LIN {X 0,Y 411.168,Z 328.267,A -85,B 0,C 180,E1 -10479.721,E2 -10479.721} C_VEL
LIN {X 0,Y 411.16,Z 328.272,A -85,B 0,C 180,E1 -10483.136,E2 -10483.136} C_VEL
LIN {X 0,Y 411.167,Z 328.27,A -85,B 0,C 180,E1 -10485.881,E2 -10485.881} C_VEL
LIN {X 0,Y 411.213,Z 328.29,A -85,B 0,C 180,E1 -10488.764,E2 -10488.764} C_VEL
LIN {X 0,Y 412.183,Z 333.965,A -85,B 0,C 180,E1 -10492.134,E2 -10492.134} C_VEL
LIN {X 0,Y 412.545,Z 338.866,A -85,B 0,C 180,E1 -10494.857,E2 -10494.857} C_VEL
LIN {X 0,Y 412.139,Z 345.061,A -85,B 0,C 180,E1 -10498.087,E2 -10498.087} C_VEL
LIN {X 0,Y 411.71,Z 351.771,A -85,B 0,C 180,E1 -10501.447,E2 -10501.447} C_VEL
LIN {X 0,Y 411.267,Z 358.916,A -85,B 0,C 180,E1 -10504.918,E2 -10504.918} C_VEL
LIN {X 0,Y 410.904,Z 366.234,A -85,B 0,C 180,E1 -10508.424,E2 -10508.424} C_VEL
LIN {X 0,Y 410.611,Z 372.815,A -85,B 0,C 180,E1 -10511.54,E2 -10511.54} C_VEL
LIN {X 0,Y 410.564,Z 374.685,A -85,B 0,C 180,E1 -10512.421,E2 -10512.421} C_VEL
LIN {X 0,Y 412.967,Z 388.008,A -85,B 0,C 180,E1 -10512.93,E2 -10512.93} C_VEL
LIN {X 0,Y 414.869,Z 400.705,A -85,B 0,C 180,E1 -10513.605,E2 -10513.605} C_VEL
LIN {X 0,Y 414.575,Z 409.621,A -85,B 0,C 180,E1 -10514.141,E2 -10514.141} C_VEL
LIN {X 0,Y 413.832,Z 420.921,A -85,B 0,C 180,E1 -10514.99,E2 -10514.99} C_VEL
LIN {X 0,Y 413.057,Z 432.111,A -85,B 0,C 180,E1 -10516.055,E2 -10516.055} C_VEL
LIN {X 0,Y 412.36,Z 441.79,A -85,B 0,C 180,E1 -10517.199,E2 -10517.199} C_VEL
LIN {X 0,Y 411.629,Z 450.278,A -85,B 0,C 180,E1 -10518.427,E2 -10518.427} C_VEL
LIN {X 0,Y 411.026,Z 458.564,A -85,B 0,C 180,E1 -10519.906,E2 -10519.906} C_VEL
LIN {X 0,Y 410.576,Z 465.244,A -85,B 0,C 180,E1 -10521.386,E2 -10521.386} C_VEL
LIN {X 0,Y 410.253,Z 471.36,A -85,B 0,C 180,E1 -10523.112,E2 -10523.112} C_VEL
LIN {X 0,Y 410.065,Z 475.333,A -85,B 0,C 180,E1 -10524.591,E2 -10524.591} C_VEL
LIN {X 0,Y 409.943,Z 478.268,A -85,B 0,C 180,E1 -10526.067,E2 -10526.067} C_VEL
LIN {X 0,Y 409.963,Z 480.666,A -85,B 0,C 180,E1 -10528.035,E2 -10528.035} C_VEL
LIN {X 0,Y 409.919,Z 481.275,A -85,B 0,C 180,E1 -10529.017,E2 -10529.017} C_VEL
LIN {X 0,Y 409.888,Z 481.491,A -85,B 0,C 180,E1 -10530,E2 -10530} C_VEL
LIN {X 0,Y 409.918,Z 481.275,A -85,B 0,C 180,E1 -10530.982,E2 -10530.982} C_VEL
LIN {X 0,Y 409.963,Z 480.669,A -85,B 0,C 180,E1 -10531.964,E2 -10531.964} C_VEL
LIN {X 0,Y 409.943,Z 478.274,A -85,B 0,C 180,E1 -10533.932,E2 -10533.932} C_VEL
LIN {X 0,Y 410.063,Z 475.336,A -85,B 0,C 180,E1 -10535.408,E2 -10535.408} C_VEL
LIN {X 0,Y 410.198,Z 471.359,A -85,B 0,C 180,E1 -10536.888,E2 -10536.888} C_VEL
LIN {X 0,Y 410.575,Z 465.247,A -85,B 0,C 180,E1 -10538.613,E2 -10538.613} C_VEL
LIN {X 0,Y 411.025,Z 458.568,A -85,B 0,C 180,E1 -10540.093,E2 -10540.093} C_VEL
LIN {X 0,Y 411.633,Z 450.282,A -85,B 0,C 180,E1 -10541.572,E2 -10541.572} C_VEL
LIN {X 0,Y 412.375,Z 441.796,A -85,B 0,C 180,E1 -10542.8,E2 -10542.8} C_VEL
LIN {X 0,Y 413.08,Z 431.211,A -85,B 0,C 180,E1 -10544.04,E2 -10544.04} C_VEL
LIN {X 0,Y 413.891,Z 419.499,A -85,B 0,C 180,E1 -10545.133,E2 -10545.133} C_VEL
LIN {X 0,Y 414.716,Z 407.771,A -85,B 0,C 180,E1 -10545.975,E2 -10545.975} C_VEL
LIN {X 0,Y 414.824,Z 400.648,A -85,B 0,C 180,E1 -10546.399,E2 -10546.399} C_VEL
LIN {X 0,Y 412.854,Z 387.284,A -85,B 0,C 180,E1 -10547.101,E2 -10547.101} C_VEL
LIN {X 0,Y 410.564,Z 374.685,A -85,B 0,C 180,E1 -10547.578,E2 -10547.578} C_VEL
LIN {X 0,Y 410.855,Z 367.344,A -85,B 0,C 180,E1 -10551.051,E2 -10551.051} C_VEL
LIN {X 0,Y 411.168,Z 360.704,A -85,B 0,C 180,E1 -10554.218,E2 -10554.218} C_VEL
LIN {X 0,Y 411.55,Z 353.989,A -85,B 0,C 180,E1 -10557.455,E2 -10557.455} C_VEL
LIN {X 0,Y 411.993,Z 347.272,A -85,B 0,C 180,E1 -10560.78,E2 -10560.78} C_VEL
LIN {X 0,Y 412.444,Z 340.595,A -85,B 0,C 180,E1 -10564.215,E2 -10564.215} C_VEL
LIN {X 0,Y 412.503,Z 337.275,A -85,B 0,C 180,E1 -10565.999,E2 -10565.999} C_VEL
LIN {X 0,Y 412.086,Z 333.137,A -85,B 0,C 180,E1 -10568.324,E2 -10568.324} C_VEL
LIN {X 0,Y 411.243,Z 328.265,A -85,B 0,C 180,E1 -10571.241,E2 -10571.241} C_VEL
LIN {X 0,Y 411.223,Z 328.263,A -85,B 0,C 180,E1 -10574.482,E2 -10574.482} C_VEL
LIN {X 0,Y 411.157,Z 328.268,A -85,B 0,C 180,E1 -10578.192,E2 -10578.192} C_VEL
LIN {X 0,Y 411.193,Z 328.263,A -85,B 0,C 180,E1 -10581.832,E2 -10581.832} C_VEL
LIN {X 0,Y 411.204,Z 328.264,A -85,B 0,C 180,E1 -10585.121,E2 -10585.121} C_VEL
LIN {X 0,Y 411.158,Z 328.269,A -85,B 0,C 180,E1 -10588.002,E2 -10588.002} C_VEL
LIN {X 0,Y 411.171,Z 328.265,A -85,B 0,C 180,E1 -10591.406,E2 -10591.406} C_VEL
LIN {X 0,Y 411.218,Z 328.261,A -85,B 0,C 180,E1 -10594.929,E2 -10594.929} C_VEL
LIN {X 0,Y 411.196,Z 328.265,A -85,B 0,C 180,E1 -10597.913,E2 -10597.913} C_VEL
LIN {X 0,Y 411.215,Z 328.261,A -85,B 0,C 180,E1 -10601.051,E2 -10601.051} C_VEL
LIN {X 0,Y 411.244,Z 328.261,A -85,B 0,C 180,E1 -10604.131,E2 -10604.131} C_VEL
LIN {X 0,Y 411.293,Z 328.25,A -85,B 0,C 180,E1 -10607.165,E2 -10607.165} C_VEL
LIN {X 0,Y 411.283,Z 328.255,A -85,B 0,C 180,E1 -10610.161,E2 -10610.161} C_VEL
LIN {X 0,Y 411.453,Z 328.231,A -85,B 0,C 180,E1 -10613.133,E2 -10613.133} C_VEL
LIN {X 0,Y 411.309,Z 328.249,A -85,B 0,C 180,E1 -10615.099,E2 -10615.099} C_VEL
LIN {X 0,Y 411.502,Z 328.228,A -85,B 0,C 180,E1 -10618.043,E2 -10618.043} C_VEL
LIN {X 0,Y 411.622,Z 328.212,A -85,B 0,C 180,E1 -10620,E2 -10620} C_VEL
LIN {X 0,Y 411.449,Z 328.231,A -85,B 0,C 180,E1 -10622.937,E2 -10622.937} C_VEL
LIN {X 0,Y 411.452,Z 328.232,A -85,B 0,C 180,E1 -10626.867,E2 -10626.867} C_VEL
LIN {X 0,Y 411.283,Z 328.254,A -85,B 0,C 180,E1 -10629.839,E2 -10629.839} C_VEL
LIN {X 0,Y 411.295,Z 328.253,A -85,B 0,C 180,E1 -10633.104,E2 -10633.104} C_VEL
LIN {X 0,Y 411.248,Z 328.258,A -85,B 0,C 180,E1 -10636.889,E2 -10636.889} C_VEL
LIN {X 0,Y 411.222,Z 328.259,A -85,B 0,C 180,E1 -10639.987,E2 -10639.987} C_VEL
LIN {X 0,Y 411.193,Z 328.267,A -85,B 0,C 180,E1 -10643.148,E2 -10643.148} C_VEL
LIN {X 0,Y 411.177,Z 328.266,A -85,B 0,C 180,E1 -10646.385,E2 -10646.385} C_VEL
LIN {X 0,Y 411.189,Z 328.263,A -85,B 0,C 180,E1 -10649.714,E2 -10649.714} C_VEL
LIN {X 0,Y 411.199,Z 328.265,A -85,B 0,C 180,E1 -10653.157,E2 -10653.157} C_VEL
LIN {X 0,Y 411.186,Z 328.268,A -85,B 0,C 180,E1 -10656.553,E2 -10656.553} C_VEL
LIN {X 0,Y 411.163,Z 328.267,A -85,B 0,C 180,E1 -10659.721,E2 -10659.721} C_VEL
LIN {X 0,Y 411.158,Z 328.268,A -85,B 0,C 180,E1 -10663.136,E2 -10663.136} C_VEL
LIN {X 0,Y 411.163,Z 328.267,A -85,B 0,C 180,E1 -10665.882,E2 -10665.882} C_VEL
LIN {X 0,Y 411.197,Z 328.265,A -85,B 0,C 180,E1 -10668.767,E2 -10668.767} C_VEL
LIN {X 0,Y 411.193,Z 328.267,A -85,B 0,C 180,E1 -10672.028,E2 -10672.028} C_VEL
LIN {X 0,Y 411.147,Z 328.274,A -85,B 0,C 180,E1 -10673.457,E2 -10673.457} C_VEL
LIN {X 0,Y 411.083,Z 328.68,A -85,B 0,C 180,E1 -10674.461,E2 -10674.461} C_VEL
LIN {X 0,Y 411.069,Z 331.626,A -85,B 0,C 180,E1 -10676.903,E2 -10676.903} C_VEL
LIN {X 0,Y 410.849,Z 335.82,A -85,B 0,C 180,E1 -10680.26,E2 -10680.26} C_VEL
LIN {X 0,Y 410.661,Z 340.084,A -85,B 0,C 180,E1 -10683.58,E2 -10683.58} C_VEL
LIN {X 0,Y 410.515,Z 344.369,A -85,B 0,C 180,E1 -10686.812,E2 -10686.812} C_VEL
LIN {X 0,Y 410.383,Z 349.289,A -85,B 0,C 180,E1 -10690.374,E2 -10690.374} C_VEL
LIN {X 0,Y 410.314,Z 352.471,A -85,B 0,C 180,E1 -10692.493,E2 -10692.493} C_VEL
LIN {X 0,Y 413.528,Z 365.928,A -85,B 0,C 180,E1 -10693.083,E2 -10693.083} C_VEL
LIN {X 0,Y 415.374,Z 375.743,A -85,B 0,C 180,E1 -10693.63,E2 -10693.63} C_VEL
LIN {X 0,Y 414.752,Z 388.201,A -85,B 0,C 180,E1 -10694.396,E2 -10694.396} C_VEL
LIN {X 0,Y 414.048,Z 398.961,A -85,B 0,C 180,E1 -10695.25,E2 -10695.25} C_VEL
LIN {X 0,Y 413.36,Z 409.923,A -85,B 0,C 180,E1 -10696.356,E2 -10696.356} C_VEL
LIN {X 0,Y 412.474,Z 420.598,A -85,B 0,C 180,E1 -10697.703,E2 -10697.703} C_VEL
LIN {X 0,Y 411.863,Z 428.466,A -85,B 0,C 180,E1 -10698.933,E2 -10698.933} C_VEL
LIN {X 0,Y 411.231,Z 436.156,A -85,B 0,C 180,E1 -10700.409,E2 -10700.409} C_VEL
LIN {X 0,Y 410.669,Z 443.213,A -85,B 0,C 180,E1 -10702.132,E2 -10702.132} C_VEL
LIN {X 0,Y 410.4,Z 447.969,A -85,B 0,C 180,E1 -10703.63,E2 -10703.63} C_VEL
LIN {X 0,Y 410.172,Z 451.508,A -85,B 0,C 180,E1 -10705.086,E2 -10705.086} C_VEL
LIN {X 0,Y 410.063,Z 453.368,A -85,B 0,C 180,E1 -10706.069,E2 -10706.069} C_VEL
LIN {X 0,Y 410.062,Z 454.765,A -85,B 0,C 180,E1 -10707.053,E2 -10707.053} C_VEL
LIN {X 0,Y 410.013,Z 455.761,A -85,B 0,C 180,E1 -10708.036,E2 -10708.036} C_VEL
LIN {X 0,Y 409.927,Z 456.609,A -85,B 0,C 180,E1 -10710,E2 -10710} C_VEL
LIN {X 0,Y 409.939,Z 456.42,A -85,B 0,C 180,E1 -10710.983,E2 -10710.983} C_VEL
LIN {X 0,Y 410.013,Z 455.835,A -85,B 0,C 180,E1 -10711.965,E2 -10711.965} C_VEL
LIN {X 0,Y 410.061,Z 454.869,A -85,B 0,C 180,E1 -10712.948,E2 -10712.948} C_VEL
LIN {X 0,Y 410.06,Z 453.516,A -85,B 0,C 180,E1 -10713.931,E2 -10713.931} C_VEL
LIN {X 0,Y 410.277,Z 450.65,A -85,B 0,C 180,E1 -10715.406,E2 -10715.406} C_VEL
LIN {X 0,Y 410.463,Z 446.768,A -85,B 0,C 180,E1 -10716.884,E2 -10716.884} C_VEL
LIN {X 0,Y 410.801,Z 441.757,A -85,B 0,C 180,E1 -10718.362,E2 -10718.362} C_VEL
LIN {X 0,Y 410.999,Z 439.011,A -85,B 0,C 180,E1 -10719.045,E2 -10719.045} C_VEL
LIN {X 0,Y 410.59,Z 436.033,A -85,B 0,C 180,E1 -10719.756,E2 -10719.756} C_VEL
LIN {X 0,Y 408.194,Z 430.826,A -85,B 0,C 180,E1 -10720.891,E2 -10720.891} C_VEL
LIN {X 0,Y 405.855,Z 424.967,A -85,B 0,C 180,E1 -10721.971,E2 -10721.971} C_VEL
LIN {X 0,Y 405.532,Z 420.966,A -85,B 0,C 180,E1 -10722.585,E2 -10722.585} C_VEL
LIN {X 0,Y 406.417,Z 410.939,A -85,B 0,C 180,E1 -10723.883,E2 -10723.883} C_VEL
LIN {X 0,Y 407.113,Z 400.203,A -85,B 0,C 180,E1 -10725.008,E2 -10725.008} C_VEL
LIN {X 0,Y 407.831,Z 389.733,A -85,B 0,C 180,E1 -10725.877,E2 -10725.877} C_VEL
LIN {X 0,Y 408.532,Z 377.621,A -85,B 0,C 180,E1 -10726.654,E2 -10726.654} C_VEL
LIN {X 0,Y 406.637,Z 367.045,A -85,B 0,C 180,E1 -10727.273,E2 -10727.273} C_VEL
LIN {X 0,Y 403.47,Z 354.02,A -85,B 0,C 180,E1 -10727.875,E2 -10727.875} C_VEL
LIN {X 0,Y 403.203,Z 352.513,A -85,B 0,C 180,E1 -10727.947,E2 -10727.947} C_VEL
LIN {X 0,Y 403.313,Z 349.051,A -85,B 0,C 180,E1 -10730.396,E2 -10730.396} C_VEL
LIN {X 0,Y 403.454,Z 344.71,A -85,B 0,C 180,E1 -10733.619,E2 -10733.619} C_VEL
LIN {X 0,Y 403.666,Z 340.39,A -85,B 0,C 180,E1 -10736.915,E2 -10736.915} C_VEL
LIN {X 0,Y 403.846,Z 336.129,A -85,B 0,C 180,E1 -10740.31,E2 -10740.31} C_VEL
LIN {X 0,Y 404.05,Z 332.333,A -85,B 0,C 180,E1 -10743.394,E2 -10743.394} C_VEL
LIN {X 0,Y 404.099,Z 330.186,A -85,B 0,C 180,E1 -10745.173,E2 -10745.173} C_VEL
LIN {X 0,Y 404.063,Z 329.158,A -85,B 0,C 180,E1 -10746.254,E2 -10746.254} C_VEL
LIN {X 0,Y 404.149,Z 329.146,A -85,B 0,C 180,E1 -10748.757,E2 -10748.757} C_VEL
LIN {X 0,Y 404.123,Z 329.148,A -85,B 0,C 180,E1 -10751.599,E2 -10751.599} C_VEL
LIN {X 0,Y 404.145,Z 329.14,A -85,B 0,C 180,E1 -10754.522,E2 -10754.522} C_VEL
LIN {X 0,Y 404.119,Z 329.147,A -85,B 0,C 180,E1 -10757.293,E2 -10757.293} C_VEL
LIN {X 0,Y 404.131,Z 329.144,A -85,B 0,C 180,E1 -10759.951,E2 -10759.951} C_VEL
LIN {X 0,Y 404.134,Z 329.146,A -85,B 0,C 180,E1 -10763.125,E2 -10763.125} C_VEL
LIN {X 0,Y 404.143,Z 329.141,A -85,B 0,C 180,E1 -10766.187,E2 -10766.187} C_VEL
LIN {X 0,Y 404.141,Z 329.142,A -85,B 0,C 180,E1 -10769.714,E2 -10769.714} C_VEL
LIN {X 0,Y 404.122,Z 329.148,A -85,B 0,C 180,E1 -10773.117,E2 -10773.117} C_VEL
LIN {X 0,Y 404.158,Z 329.14,A -85,B 0,C 180,E1 -10776.425,E2 -10776.425} C_VEL
LIN {X 0,Y 404.188,Z 329.135,A -85,B 0,C 180,E1 -10779.874,E2 -10779.874} C_VEL
LIN {X 0,Y 404.213,Z 329.136,A -85,B 0,C 180,E1 -10782.993,E2 -10782.993} C_VEL
LIN {X 0,Y 404.279,Z 329.127,A -85,B 0,C 180,E1 -10786.939,E2 -10786.939} C_VEL
LIN {X 0,Y 404.254,Z 329.128,A -85,B 0,C 180,E1 -10789.988,E2 -10789.988} C_VEL
LIN {X 0,Y 404.408,Z 329.11,A -85,B 0,C 180,E1 -10793.013,E2 -10793.013} C_VEL
LIN {X 0,Y 404.28,Z 329.125,A -85,B 0,C 180,E1 -10795.013,E2 -10795.013} C_VEL
LIN {X 0,Y 404.475,Z 329.101,A -85,B 0,C 180,E1 -10798.008,E2 -10798.008} C_VEL
LIN {X 0,Y 404.595,Z 329.087,A -85,B 0,C 180,E1 -10800,E2 -10800} C_VEL
LIN {X 0,Y 404.411,Z 329.108,A -85,B 0,C 180,E1 -10802.988,E2 -10802.988} C_VEL
LIN {X 0,Y 404.42,Z 329.111,A -85,B 0,C 180,E1 -10805.985,E2 -10805.985} C_VEL
LIN {X 0,Y 404.287,Z 329.123,A -85,B 0,C 180,E1 -10809.001,E2 -10809.001} C_VEL
LIN {X 0,Y 404.252,Z 329.133,A -85,B 0,C 180,E1 -10812.042,E2 -10812.042} C_VEL
LIN {X 0,Y 404.199,Z 329.134,A -85,B 0,C 180,E1 -10815.118,E2 -10815.118} C_VEL
LIN {X 0,Y 404.206,Z 329.136,A -85,B 0,C 180,E1 -10818.238,E2 -10818.238} C_VEL
LIN {X 0,Y 404.135,Z 329.145,A -85,B 0,C 180,E1 -10821.42,E2 -10821.42} C_VEL
LIN {X 0,Y 404.163,Z 329.138,A -85,B 0,C 180,E1 -10824.667,E2 -10824.667} C_VEL
LIN {X 0,Y 404.116,Z 329.146,A -85,B 0,C 180,E1 -10828.006,E2 -10828.006} C_VEL
LIN {X 0,Y 404.14,Z 329.142,A -85,B 0,C 180,E1 -10830.286,E2 -10830.286} C_VEL
LIN {X 0,Y 404.143,Z 329.144,A -85,B 0,C 180,E1 -10833.813,E2 -10833.813} C_VEL
LIN {X 0,Y 404.136,Z 329.144,A -85,B 0,C 180,E1 -10836.876,E2 -10836.876} C_VEL
LIN {X 0,Y 404.115,Z 329.144,A -85,B 0,C 180,E1 -10840.075,E2 -10840.075} C_VEL
LIN {X 0,Y 404.14,Z 329.147,A -85,B 0,C 180,E1 -10843.082,E2 -10843.082} C_VEL
LIN {X 0,Y 404.147,Z 329.145,A -85,B 0,C 180,E1 -10845.926,E2 -10845.926} C_VEL
LIN {X 0,Y 404.169,Z 329.157,A -85,B 0,C 180,E1 -10848.476,E2 -10848.476} C_VEL
LIN {X 0,Y 404.99,Z 333.851,A -85,B 0,C 180,E1 -10851.344,E2 -10851.344} C_VEL
LIN {X 0,Y 405.502,Z 338.276,A -85,B 0,C 180,E1 -10853.895,E2 -10853.895} C_VEL
LIN {X 0,Y 405.331,Z 342.775,A -85,B 0,C 180,E1 -10856.333,E2 -10856.333} C_VEL
LIN {X 0,Y 404.905,Z 349.379,A -85,B 0,C 180,E1 -10859.778,E2 -10859.778} C_VEL
LIN {X 0,Y 404.427,Z 356.085,A -85,B 0,C 180,E1 -10863.14,E2 -10863.14} C_VEL
LIN {X 0,Y 404.036,Z 362.738,A -85,B 0,C 180,E1 -10866.417,E2 -10866.417} C_VEL
LIN {X 0,Y 403.676,Z 370.283,A -85,B 0,C 180,E1 -10870.076,E2 -10870.076} C_VEL
LIN {X 0,Y 403.508,Z 374.603,A -85,B 0,C 180,E1 -10872.107,E2 -10872.107} C_VEL
LIN {X 0,Y 405.943,Z 387.743,A -85,B 0,C 180,E1 -10872.624,E2 -10872.624} C_VEL
LIN {X 0,Y 407.939,Z 401.142,A -85,B 0,C 180,E1 -10873.356,E2 -10873.356} C_VEL
LIN {X 0,Y 407.839,Z 407.78,A -85,B 0,C 180,E1 -10873.761,E2 -10873.761} C_VEL
LIN {X 0,Y 407.063,Z 419.278,A -85,B 0,C 180,E1 -10874.606,E2 -10874.606} C_VEL
LIN {X 0,Y 406.231,Z 430.438,A -85,B 0,C 180,E1 -10875.657,E2 -10875.657} C_VEL
LIN {X 0,Y 405.543,Z 439.624,A -85,B 0,C 180,E1 -10876.725,E2 -10876.725} C_VEL
LIN {X 0,Y 404.791,Z 448.476,A -85,B 0,C 180,E1 -10877.974,E2 -10877.974} C_VEL
LIN {X 0,Y 404.139,Z 457.112,A -85,B 0,C 180,E1 -10879.479,E2 -10879.479} C_VEL
LIN {X 0,Y 403.603,Z 464.015,A -85,B 0,C 180,E1 -10880.983,E2 -10880.983} C_VEL
LIN {X 0,Y 403.212,Z 469.548,A -85,B 0,C 180,E1 -10882.488,E2 -10882.488} C_VEL
LIN {X 0,Y 402.999,Z 473.89,A -85,B 0,C 180,E1 -10883.994,E2 -10883.994} C_VEL
LIN {X 0,Y 402.973,Z 476.191,A -85,B 0,C 180,E1 -10884.997,E2 -10884.997} C_VEL
LIN {X 0,Y 402.865,Z 478.053,A -85,B 0,C 180,E1 -10885.998,E2 -10885.998} C_VEL
LIN {X 0,Y 402.861,Z 480.451,A -85,B 0,C 180,E1 -10888,E2 -10888} C_VEL
LIN {X 0,Y 402.847,Z 481.06,A -85,B 0,C 180,E1 -10889,E2 -10889} C_VEL
LIN {X 0,Y 402.814,Z 481.276,A -85,B 0,C 180,E1 -10890,E2 -10890} C_VEL
LIN {X 0,Y 402.847,Z 481.061,A -85,B 0,C 180,E1 -10890.999,E2 -10890.999} C_VEL
LIN {X 0,Y 402.861,Z 480.453,A -85,B 0,C 180,E1 -10891.999,E2 -10891.999} C_VEL
LIN {X 0,Y 402.865,Z 478.058,A -85,B 0,C 180,E1 -10894.001,E2 -10894.001} C_VEL
LIN {X 0,Y 402.966,Z 475.12,A -85,B 0,C 180,E1 -10895.504,E2 -10895.504} C_VEL
LIN {X 0,Y 403.117,Z 471.142,A -85,B 0,C 180,E1 -10897.009,E2 -10897.009} C_VEL
LIN {X 0,Y 403.534,Z 465.03,A -85,B 0,C 180,E1 -10898.765,E2 -10898.765} C_VEL
LIN {X 0,Y 404.022,Z 458.351,A -85,B 0,C 180,E1 -10900.27,E2 -10900.27} C_VEL
LIN {X 0,Y 404.654,Z 450.065,A -85,B 0,C 180,E1 -10901.775,E2 -10901.775} C_VEL
LIN {X 0,Y 405.418,Z 441.577,A -85,B 0,C 180,E1 -10903.023,E2 -10903.023} C_VEL
LIN {X 0,Y 406.147,Z 430.883,A -85,B 0,C 180,E1 -10904.297,E2 -10904.297} C_VEL
LIN {X 0,Y 407.021,Z 419.28,A -85,B 0,C 180,E1 -10905.395,E2 -10905.395} C_VEL
LIN {X 0,Y 407.87,Z 407.777,A -85,B 0,C 180,E1 -10906.236,E2 -10906.236} C_VEL
LIN {X 0,Y 408.031,Z 402.165,A -85,B 0,C 180,E1 -10906.581,E2 -10906.581} C_VEL
LIN {X 0,Y 406.151,Z 389.01,A -85,B 0,C 180,E1 -10907.312,E2 -10907.312} C_VEL
LIN {X 0,Y 403.705,Z 376.012,A -85,B 0,C 180,E1 -10907.852,E2 -10907.852} C_VEL
LIN {X 0,Y 403.488,Z 374.444,A -85,B 0,C 180,E1 -10907.91,E2 -10907.91} C_VEL
LIN {X 0,Y 403.81,Z 367.158,A -85,B 0,C 180,E1 -10911.437,E2 -10911.437} C_VEL
LIN {X 0,Y 404.163,Z 360.53,A -85,B 0,C 180,E1 -10914.666,E2 -10914.666} C_VEL
LIN {X 0,Y 404.568,Z 353.836,A -85,B 0,C 180,E1 -10917.971,E2 -10917.971} C_VEL
LIN {X 0,Y 405.025,Z 347.129,A -85,B 0,C 180,E1 -10921.369,E2 -10921.369} C_VEL
LIN {X 0,Y 405.496,Z 340.468,A -85,B 0,C 180,E1 -10924.885,E2 -10924.885} C_VEL
LIN {X 0,Y 405.344,Z 336.503,A -85,B 0,C 180,E1 -10927.102,E2 -10927.102} C_VEL
LIN {X 0,Y 404.606,Z 331.34,A -85,B 0,C 180,E1 -10930.157,E2 -10930.157} C_VEL
LIN {X 0,Y 404.212,Z 329.142,A -85,B 0,C 180,E1 -10931.614,E2 -10931.614} C_VEL
LIN {X 0,Y 404.187,Z 329.14,A -85,B 0,C 180,E1 -10934.528,E2 -10934.528} C_VEL
LIN {X 0,Y 404.118,Z 329.145,A -85,B 0,C 180,E1 -10937.293,E2 -10937.293} C_VEL
LIN {X 0,Y 404.125,Z 329.142,A -85,B 0,C 180,E1 -10939.95,E2 -10939.95} C_VEL
LIN {X 0,Y 404.131,Z 329.145,A -85,B 0,C 180,E1 -10943.124,E2 -10943.124} C_VEL
LIN {X 0,Y 404.138,Z 329.144,A -85,B 0,C 180,E1 -10946.187,E2 -10946.187} C_VEL
LIN {X 0,Y 404.135,Z 329.142,A -85,B 0,C 180,E1 -10949.714,E2 -10949.714} C_VEL
LIN {X 0,Y 404.119,Z 329.143,A -85,B 0,C 180,E1 -10953.117,E2 -10953.117} C_VEL
LIN {X 0,Y 404.157,Z 329.143,A -85,B 0,C 180,E1 -10956.425,E2 -10956.425} C_VEL
LIN {X 0,Y 404.182,Z 329.139,A -85,B 0,C 180,E1 -10959.874,E2 -10959.874} C_VEL
LIN {X 0,Y 404.206,Z 329.133,A -85,B 0,C 180,E1 -10962.993,E2 -10962.993} C_VEL
LIN {X 0,Y 404.273,Z 329.124,A -85,B 0,C 180,E1 -10966.939,E2 -10966.939} C_VEL
LIN {X 0,Y 404.248,Z 329.133,A -85,B 0,C 180,E1 -10969.988,E2 -10969.988} C_VEL
LIN {X 0,Y 404.404,Z 329.109,A -85,B 0,C 180,E1 -10973.013,E2 -10973.013} C_VEL
LIN {X 0,Y 404.281,Z 329.124,A -85,B 0,C 180,E1 -10975.014,E2 -10975.014} C_VEL
LIN {X 0,Y 404.472,Z 329.104,A -85,B 0,C 180,E1 -10978.009,E2 -10978.009} C_VEL
LIN {X 0,Y 404.591,Z 329.088,A -85,B 0,C 180,E1 -10980,E2 -10980} C_VEL
LIN {X 0,Y 404.407,Z 329.108,A -85,B 0,C 180,E1 -10982.989,E2 -10982.989} C_VEL
LIN {X 0,Y 404.403,Z 329.11,A -85,B 0,C 180,E1 -10986.987,E2 -10986.987} C_VEL
LIN {X 0,Y 404.249,Z 329.129,A -85,B 0,C 180,E1 -10990.012,E2 -10990.012} C_VEL
LIN {X 0,Y 404.257,Z 329.131,A -85,B 0,C 180,E1 -10993.212,E2 -10993.212} C_VEL
LIN {X 0,Y 404.207,Z 329.136,A -85,B 0,C 180,E1 -10997.008,E2 -10997.008} C_VEL
LIN {X 0,Y 404.155,Z 329.14,A -85,B 0,C 180,E1 -11000.352,E2 -11000.352} C_VEL
LIN {X 0,Y 404.157,Z 329.141,A -85,B 0,C 180,E1 -11003.575,E2 -11003.575} C_VEL
LIN {X 0,Y 404.119,Z 329.148,A -85,B 0,C 180,E1 -11006.883,E2 -11006.883} C_VEL
LIN {X 0,Y 404.136,Z 329.142,A -85,B 0,C 180,E1 -11010.286,E2 -11010.286} C_VEL
LIN {X 0,Y 404.138,Z 329.141,A -85,B 0,C 180,E1 -11013.813,E2 -11013.813} C_VEL
LIN {X 0,Y 404.129,Z 329.147,A -85,B 0,C 180,E1 -11016.876,E2 -11016.876} C_VEL
LIN {X 0,Y 404.11,Z 329.146,A -85,B 0,C 180,E1 -11020.076,E2 -11020.076} C_VEL
LIN {X 0,Y 404.138,Z 329.142,A -85,B 0,C 180,E1 -11023.083,E2 -11023.083} C_VEL
LIN {X 0,Y 404.143,Z 329.141,A -85,B 0,C 180,E1 -11025.927,E2 -11025.927} C_VEL
LIN {X 0,Y 404.148,Z 329.144,A -85,B 0,C 180,E1 -11028.64,E2 -11028.64} C_VEL
LIN {X 0,Y 404.154,Z 329.14,A -85,B 0,C 180,E1 -11031.493,E2 -11031.493} C_VEL
LIN {X 0,Y 404.056,Z 329.156,A -85,B 0,C 180,E1 -11033.746,E2 -11033.746} C_VEL
LIN {X 0,Y 404.083,Z 330.258,A -85,B 0,C 180,E1 -11034.975,E2 -11034.975} C_VEL
LIN {X 0,Y 404.009,Z 333.112,A -85,B 0,C 180,E1 -11037.368,E2 -11037.368} C_VEL
LIN {X 0,Y 403.781,Z 337.412,A -85,B 0,C 180,E1 -11040.834,E2 -11040.834} C_VEL
LIN {X 0,Y 403.565,Z 341.679,A -85,B 0,C 180,E1 -11044.192,E2 -11044.192} C_VEL
LIN {X 0,Y 403.418,Z 346.003,A -85,B 0,C 180,E1 -11047.465,E2 -11047.465} C_VEL
LIN {X 0,Y 403.298,Z 350.402,A -85,B 0,C 180,E1 -11050.665,E2 -11050.665} C_VEL
LIN {X 0,Y 403.248,Z 352.55,A -85,B 0,C 180,E1 -11052.172,E2 -11052.172} C_VEL
LIN {X 0,Y 406.438,Z 365.869,A -85,B 0,C 180,E1 -11052.766,E2 -11052.766} C_VEL
LIN {X 0,Y 408.525,Z 376.745,A -85,B 0,C 180,E1 -11053.392,E2 -11053.392} C_VEL
LIN {X 0,Y 407.918,Z 388.423,A -85,B 0,C 180,E1 -11054.128,E2 -11054.128} C_VEL
LIN {X 0,Y 407.191,Z 399.182,A -85,B 0,C 180,E1 -11054.996,E2 -11054.996} C_VEL
LIN {X 0,Y 406.47,Z 410.142,A -85,B 0,C 180,E1 -11056.12,E2 -11056.12} C_VEL
LIN {X 0,Y 405.55,Z 420.816,A -85,B 0,C 180,E1 -11057.49,E2 -11057.49} C_VEL
LIN {X 0,Y 404.911,Z 428.683,A -85,B 0,C 180,E1 -11058.74,E2 -11058.74} C_VEL
LIN {X 0,Y 404.242,Z 436.374,A -85,B 0,C 180,E1 -11060.241,E2 -11060.241} C_VEL
LIN {X 0,Y 403.628,Z 443.43,A -85,B 0,C 180,E1 -11061.993,E2 -11061.993} C_VEL
LIN {X 0,Y 403.35,Z 447.581,A -85,B 0,C 180,E1 -11063.303,E2 -11063.303} C_VEL
LIN {X 0,Y 403.116,Z 451.724,A -85,B 0,C 180,E1 -11065,E2 -11065} C_VEL
LIN {X 0,Y 402.98,Z 453.584,A -85,B 0,C 180,E1 -11066,E2 -11066} C_VEL
LIN {X 0,Y 402.966,Z 454.982,A -85,B 0,C 180,E1 -11067.001,E2 -11067.001} C_VEL
LIN {X 0,Y 402.945,Z 455.976,A -85,B 0,C 180,E1 -11068.001,E2 -11068.001} C_VEL
LIN {X 0,Y 402.851,Z 456.824,A -85,B 0,C 180,E1 -11070,E2 -11070} C_VEL
LIN {X 0,Y 402.867,Z 456.635,A -85,B 0,C 180,E1 -11071,E2 -11071} C_VEL
LIN {X 0,Y 402.945,Z 456.049,A -85,B 0,C 180,E1 -11071.999,E2 -11071.999} C_VEL
LIN {X 0,Y 402.965,Z 455.084,A -85,B 0,C 180,E1 -11073,E2 -11073} C_VEL
LIN {X 0,Y 402.977,Z 453.731,A -85,B 0,C 180,E1 -11074.001,E2 -11074.001} C_VEL
LIN {X 0,Y 403.226,Z 450.864,A -85,B 0,C 180,E1 -11075.501,E2 -11075.501} C_VEL
LIN {X 0,Y 403.404,Z 446.983,A -85,B 0,C 180,E1 -11077.005,E2 -11077.005} C_VEL
LIN {X 0,Y 403.772,Z 441.971,A -85,B 0,C 180,E1 -11078.508,E2 -11078.508} C_VEL
LIN {X 0,Y 404.319,Z 435.661,A -85,B 0,C 180,E1 -11080.01,E2 -11080.01} C_VEL
LIN {X 0,Y 404.968,Z 427.761,A -85,B 0,C 180,E1 -11081.512,E2 -11081.512} C_VEL
LIN {X 0,Y 405.532,Z 420.966,A -85,B 0,C 180,E1 -11082.585,E2 -11082.585} C_VEL
LIN {X 0,Y 405.229,Z 416.856,A -85,B 0,C 180,E1 -11083.178,E2 -11083.178} C_VEL
LIN {X 0,Y 401.963,Z 407.086,A -85,B 0,C 180,E1 -11084.506,E2 -11084.506} C_VEL
LIN {X 0,Y 400.516,Z 401.003,A -85,B 0,C 180,E1 -11085.2,E2 -11085.2} C_VEL
LIN {X 0,Y 400.425,Z 397.716,A -85,B 0,C 180,E1 -11085.515,E2 -11085.515} C_VEL
LIN {X 0,Y 401.278,Z 386.712,A -85,B 0,C 180,E1 -11086.383,E2 -11086.383} C_VEL
LIN {X 0,Y 401.727,Z 378.448,A -85,B 0,C 180,E1 -11086.909,E2 -11086.909} C_VEL
LIN {X 0,Y 399.631,Z 367.095,A -85,B 0,C 180,E1 -11087.592,E2 -11087.592} C_VEL
LIN {X 0,Y 396.272,Z 353.536,A -85,B 0,C 180,E1 -11088.231,E2 -11088.231} C_VEL
LIN {X 0,Y 396.148,Z 352.696,A -85,B 0,C 180,E1 -11088.288,E2 -11088.288} C_VEL
LIN {X 0,Y 396.248,Z 349.252,A -85,B 0,C 180,E1 -11090.777,E2 -11090.777} C_VEL
LIN {X 0,Y 396.433,Z 344.892,A -85,B 0,C 180,E1 -11094.063,E2 -11094.063} C_VEL
LIN {X 0,Y 396.651,Z 340.306,A -85,B 0,C 180,E1 -11097.635,E2 -11097.635} C_VEL
LIN {X 0,Y 396.844,Z 336.279,A -85,B 0,C 180,E1 -11100.903,E2 -11100.903} C_VEL
LIN {X 0,Y 397.012,Z 332.895,A -85,B 0,C 180,E1 -11103.694,E2 -11103.694} C_VEL
LIN {X 0,Y 397.02,Z 330.488,A -85,B 0,C 180,E1 -11105.744,E2 -11105.744} C_VEL
LIN {X 0,Y 397.077,Z 330.027,A -85,B 0,C 180,E1 -11107.205,E2 -11107.205} C_VEL
LIN {X 0,Y 397.102,Z 330.018,A -85,B 0,C 180,E1 -11110.445,E2 -11110.445} C_VEL
LIN {X 0,Y 397.101,Z 330.024,A -85,B 0,C 180,E1 -11113.648,E2 -11113.648} C_VEL
LIN {X 0,Y 397.089,Z 330.019,A -85,B 0,C 180,E1 -11116.522,E2 -11116.522} C_VEL
LIN {X 0,Y 397.084,Z 330.02,A -85,B 0,C 180,E1 -11120.419,E2 -11120.419} C_VEL
LIN {X 0,Y 397.095,Z 330.022,A -85,B 0,C 180,E1 -11123.004,E2 -11123.004} C_VEL
LIN {X 0,Y 397.117,Z 330.016,A -85,B 0,C 180,E1 -11126.282,E2 -11126.282} C_VEL
LIN {X 0,Y 397.096,Z 330.018,A -85,B 0,C 180,E1 -11130.137,E2 -11130.137} C_VEL
LIN {X 0,Y 397.084,Z 330.021,A -85,B 0,C 180,E1 -11133.738,E2 -11133.738} C_VEL
LIN {X 0,Y 397.104,Z 330.022,A -85,B 0,C 180,E1 -11137.085,E2 -11137.085} C_VEL
LIN {X 0,Y 397.145,Z 330.014,A -85,B 0,C 180,E1 -11140.353,E2 -11140.353} C_VEL
LIN {X 0,Y 397.162,Z 330.01,A -85,B 0,C 180,E1 -11143.553,E2 -11143.553} C_VEL
LIN {X 0,Y 397.225,Z 330.008,A -85,B 0,C 180,E1 -11146.703,E2 -11146.703} C_VEL
LIN {X 0,Y 397.214,Z 330.004,A -85,B 0,C 180,E1 -11149.809,E2 -11149.809} C_VEL
LIN {X 0,Y 397.361,Z 329.989,A -85,B 0,C 180,E1 -11152.888,E2 -11152.888} C_VEL
LIN {X 0,Y 397.252,Z 330.001,A -85,B 0,C 180,E1 -11154.925,E2 -11154.925} C_VEL
LIN {X 0,Y 397.444,Z 329.977,A -85,B 0,C 180,E1 -11157.973,E2 -11157.973} C_VEL
LIN {X 0,Y 397.565,Z 329.963,A -85,B 0,C 180,E1 -11160,E2 -11160} C_VEL
LIN {X 0,Y 397.37,Z 329.985,A -85,B 0,C 180,E1 -11163.041,E2 -11163.041} C_VEL
LIN {X 0,Y 397.37,Z 329.989,A -85,B 0,C 180,E1 -11166.092,E2 -11166.092} C_VEL
LIN {X 0,Y 397.249,Z 329.999,A -85,B 0,C 180,E1 -11169.162,E2 -11169.162} C_VEL
LIN {X 0,Y 397.215,Z 330.007,A -85,B 0,C 180,E1 -11172.258,E2 -11172.258} C_VEL
LIN {X 0,Y 397.173,Z 330.01,A -85,B 0,C 180,E1 -11175.392,E2 -11175.392} C_VEL
LIN {X 0,Y 397.158,Z 330.011,A -85,B 0,C 180,E1 -11178.574,E2 -11178.574} C_VEL
LIN {X 0,Y 397.093,Z 330.024,A -85,B 0,C 180,E1 -11181.819,E2 -11181.819} C_VEL
LIN {X 0,Y 397.105,Z 330.018,A -85,B 0,C 180,E1 -11185.135,E2 -11185.135} C_VEL
LIN {X 0,Y 397.068,Z 330.022,A -85,B 0,C 180,E1 -11188.548,E2 -11188.548} C_VEL
LIN {X 0,Y 397.079,Z 330.024,A -85,B 0,C 180,E1 -11191.837,E2 -11191.837} C_VEL
LIN {X 0,Y 397.124,Z 330.015,A -85,B 0,C 180,E1 -11194.494,E2 -11194.494} C_VEL
LIN {X 0,Y 397.093,Z 330.019,A -85,B 0,C 180,E1 -11198.276,E2 -11198.276} C_VEL
LIN {X 0,Y 397.049,Z 330.024,A -85,B 0,C 180,E1 -11201.977,E2 -11201.977} C_VEL
LIN {X 0,Y 397.085,Z 330.025,A -85,B 0,C 180,E1 -11205.069,E2 -11205.069} C_VEL
LIN {X 0,Y 397.136,Z 330.216,A -85,B 0,C 180,E1 -11208.294,E2 -11208.294} C_VEL
LIN {X 0,Y 397.907,Z 334.547,A -85,B 0,C 180,E1 -11211,E2 -11211} C_VEL
LIN {X 0,Y 398.373,Z 338.15,A -85,B 0,C 180,E1 -11213.143,E2 -11213.143} C_VEL
LIN {X 0,Y 398.486,Z 341.468,A -85,B 0,C 180,E1 -11215.027,E2 -11215.027} C_VEL
LIN {X 0,Y 398.105,Z 347.018,A -85,B 0,C 180,E1 -11218.021,E2 -11218.021} C_VEL
LIN {X 0,Y 397.605,Z 353.69,A -85,B 0,C 180,E1 -11221.494,E2 -11221.494} C_VEL
LIN {X 0,Y 397.179,Z 360.36,A -85,B 0,C 180,E1 -11224.87,E2 -11224.87} C_VEL
LIN {X 0,Y 396.775,Z 366.97,A -85,B 0,C 180,E1 -11228.163,E2 -11228.163} C_VEL
LIN {X 0,Y 396.463,Z 373.497,A -85,B 0,C 180,E1 -11231.393,E2 -11231.393} C_VEL
LIN {X 0,Y 396.465,Z 374.393,A -85,B 0,C 180,E1 -11231.778,E2 -11231.778} C_VEL
LIN {X 0,Y 398.935,Z 387.49,A -85,B 0,C 180,E1 -11232.307,E2 -11232.307} C_VEL
LIN {X 0,Y 400.909,Z 400.557,A -85,B 0,C 180,E1 -11233.034,E2 -11233.034} C_VEL
LIN {X 0,Y 401.099,Z 406.049,A -85,B 0,C 180,E1 -11233.381,E2 -11233.381} C_VEL
LIN {X 0,Y 400.293,Z 417.526,A -85,B 0,C 180,E1 -11234.208,E2 -11234.208} C_VEL
LIN {X 0,Y 399.461,Z 428.52,A -85,B 0,C 180,E1 -11235.22,E2 -11235.22} C_VEL
LIN {X 0,Y 398.584,Z 439.409,A -85,B 0,C 180,E1 -11236.489,E2 -11236.489} C_VEL
LIN {X 0,Y 397.822,Z 448.262,A -85,B 0,C 180,E1 -11237.761,E2 -11237.761} C_VEL
LIN {X 0,Y 397.103,Z 456.896,A -85,B 0,C 180,E1 -11239.29,E2 -11239.29} C_VEL
LIN {X 0,Y 396.567,Z 463.799,A -85,B 0,C 180,E1 -11240.822,E2 -11240.822} C_VEL
LIN {X 0,Y 396.162,Z 469.332,A -85,B 0,C 180,E1 -11242.354,E2 -11242.354} C_VEL
LIN {X 0,Y 395.93,Z 473.675,A -85,B 0,C 180,E1 -11243.886,E2 -11243.886} C_VEL
LIN {X 0,Y 395.886,Z 475.975,A -85,B 0,C 180,E1 -11244.907,E2 -11244.907} C_VEL
LIN {X 0,Y 395.789,Z 477.838,A -85,B 0,C 180,E1 -11245.927,E2 -11245.927} C_VEL
LIN {X 0,Y 395.76,Z 480.235,A -85,B 0,C 180,E1 -11247.964,E2 -11247.964} C_VEL
LIN {X 0,Y 395.776,Z 480.845,A -85,B 0,C 180,E1 -11248.982,E2 -11248.982} C_VEL
LIN {X 0,Y 395.744,Z 481.061,A -85,B 0,C 180,E1 -11250,E2 -11250} C_VEL
LIN {X 0,Y 395.776,Z 480.846,A -85,B 0,C 180,E1 -11251.017,E2 -11251.017} C_VEL
LIN {X 0,Y 395.76,Z 480.237,A -85,B 0,C 180,E1 -11252.035,E2 -11252.035} C_VEL
LIN {X 0,Y 395.789,Z 477.842,A -85,B 0,C 180,E1 -11254.072,E2 -11254.072} C_VEL
LIN {X 0,Y 395.871,Z 474.903,A -85,B 0,C 180,E1 -11255.603,E2 -11255.603} C_VEL
LIN {X 0,Y 396.062,Z 470.926,A -85,B 0,C 180,E1 -11257.135,E2 -11257.135} C_VEL
LIN {X 0,Y 396.48,Z 464.813,A -85,B 0,C 180,E1 -11258.922,E2 -11258.922} C_VEL
LIN {X 0,Y 397.023,Z 458.134,A -85,B 0,C 180,E1 -11260.453,E2 -11260.453} C_VEL
LIN {X 0,Y 397.686,Z 449.847,A -85,B 0,C 180,E1 -11261.984,E2 -11261.984} C_VEL
LIN {X 0,Y 398.467,Z 441.359,A -85,B 0,C 180,E1 -11263.254,E2 -11263.254} C_VEL
LIN {X 0,Y 399.17,Z 431.58,A -85,B 0,C 180,E1 -11264.451,E2 -11264.451} C_VEL
LIN {X 0,Y 400.046,Z 420.49,A -85,B 0,C 180,E1 -11265.539,E2 -11265.539} C_VEL
LIN {X 0,Y 400.908,Z 409.365,A -85,B 0,C 180,E1 -11266.401,E2 -11266.401} C_VEL
LIN {X 0,Y 401.114,Z 402.493,A -85,B 0,C 180,E1 -11266.843,E2 -11266.843} C_VEL
LIN {X 0,Y 399.17,Z 389.013,A -85,B 0,C 180,E1 -11267.614,E2 -11267.614} C_VEL
LIN {X 0,Y 396.701,Z 375.932,A -85,B 0,C 180,E1 -11268.174,E2 -11268.174} C_VEL
LIN {X 0,Y 396.456,Z 374.242,A -85,B 0,C 180,E1 -11268.239,E2 -11268.239} C_VEL
LIN {X 0,Y 396.775,Z 366.97,A -85,B 0,C 180,E1 -11271.836,E2 -11271.836} C_VEL
LIN {X 0,Y 397.178,Z 360.357,A -85,B 0,C 180,E1 -11275.129,E2 -11275.129} C_VEL
LIN {X 0,Y 397.6,Z 353.679,A -85,B 0,C 180,E1 -11278.505,E2 -11278.505} C_VEL
LIN {X 0,Y 397.996,Z 348.096,A -85,B 0,C 180,E1 -11281.393,E2 -11281.393} C_VEL
LIN {X 0,Y 398.485,Z 341.448,A -85,B 0,C 180,E1 -11284.972,E2 -11284.972} C_VEL
LIN {X 0,Y 398.293,Z 337.14,A -85,B 0,C 180,E1 -11287.435,E2 -11287.435} C_VEL
LIN {X 0,Y 397.819,Z 333.712,A -85,B 0,C 180,E1 -11289.492,E2 -11289.492} C_VEL
LIN {X 0,Y 397.155,Z 330.018,A -85,B 0,C 180,E1 -11291.91,E2 -11291.91} C_VEL
LIN {X 0,Y 397.106,Z 330.023,A -85,B 0,C 180,E1 -11295.064,E2 -11295.064} C_VEL
LIN {X 0,Y 397.048,Z 330.024,A -85,B 0,C 180,E1 -11298.022,E2 -11298.022} C_VEL
LIN {X 0,Y 397.091,Z 330.019,A -85,B 0,C 180,E1 -11301.723,E2 -11301.723} C_VEL
LIN {X 0,Y 397.119,Z 330.016,A -85,B 0,C 180,E1 -11305.506,E2 -11305.506} C_VEL
LIN {X 0,Y 397.069,Z 330.023,A -85,B 0,C 180,E1 -11309.117,E2 -11309.117} C_VEL
LIN {X 0,Y 397.084,Z 330.024,A -85,B 0,C 180,E1 -11312.602,E2 -11312.602} C_VEL
LIN {X 0,Y 397.118,Z 330.018,A -85,B 0,C 180,E1 -11315.981,E2 -11315.981} C_VEL
LIN {X 0,Y 397.13,Z 330.016,A -85,B 0,C 180,E1 -11319.704,E2 -11319.704} C_VEL
LIN {X 0,Y 397.173,Z 330.01,A -85,B 0,C 180,E1 -11322.844,E2 -11322.844} C_VEL
LIN {X 0,Y 397.219,Z 330.003,A -85,B 0,C 180,E1 -11326.702,E2 -11326.702} C_VEL
LIN {X 0,Y 397.208,Z 330.009,A -85,B 0,C 180,E1 -11329.809,E2 -11329.809} C_VEL
LIN {X 0,Y 397.356,Z 329.986,A -85,B 0,C 180,E1 -11332.888,E2 -11332.888} C_VEL
LIN {X 0,Y 397.253,Z 329.999,A -85,B 0,C 180,E1 -11334.925,E2 -11334.925} C_VEL
LIN {X 0,Y 397.441,Z 329.98,A -85,B 0,C 180,E1 -11337.973,E2 -11337.973} C_VEL
LIN {X 0,Y 397.561,Z 329.963,A -85,B 0,C 180,E1 -11340,E2 -11340} C_VEL
LIN {X 0,Y 397.367,Z 329.985,A -85,B 0,C 180,E1 -11343.042,E2 -11343.042} C_VEL
LIN {X 0,Y 397.355,Z 329.989,A -85,B 0,C 180,E1 -11347.112,E2 -11347.112} C_VEL
LIN {X 0,Y 397.208,Z 330.005,A -85,B 0,C 180,E1 -11350.191,E2 -11350.191} C_VEL
LIN {X 0,Y 397.217,Z 330.008,A -85,B 0,C 180,E1 -11353.321,E2 -11353.321} C_VEL
LIN {X 0,Y 397.173,Z 330.014,A -85,B 0,C 180,E1 -11357.156,E2 -11357.156} C_VEL
LIN {X 0,Y 397.094,Z 330.021,A -85,B 0,C 180,E1 -11360.731,E2 -11360.731} C_VEL
LIN {X 0,Y 397.118,Z 330.016,A -85,B 0,C 180,E1 -11364.019,E2 -11364.019} C_VEL
LIN {X 0,Y 397.076,Z 330.021,A -85,B 0,C 180,E1 -11367.755,E2 -11367.755} C_VEL
LIN {X 0,Y 397.07,Z 330.027,A -85,B 0,C 180,E1 -11370.883,E2 -11370.883} C_VEL
LIN {X 0,Y 397.119,Z 330.019,A -85,B 0,C 180,E1 -11374.494,E2 -11374.494} C_VEL
LIN {X 0,Y 397.086,Z 330.022,A -85,B 0,C 180,E1 -11378.277,E2 -11378.277} C_VEL
LIN {X 0,Y 397.047,Z 330.026,A -85,B 0,C 180,E1 -11381.978,E2 -11381.978} C_VEL
LIN {X 0,Y 397.081,Z 330.021,A -85,B 0,C 180,E1 -11385.07,E2 -11385.07} C_VEL
LIN {X 0,Y 397.106,Z 330.02,A -85,B 0,C 180,E1 -11388.015,E2 -11388.015} C_VEL
LIN {X 0,Y 397.131,Z 330.014,A -85,B 0,C 180,E1 -11391.139,E2 -11391.139} C_VEL
LIN {X 0,Y 397.075,Z 330.028,A -85,B 0,C 180,E1 -11393.004,E2 -11393.004} C_VEL
LIN {X 0,Y 397.02,Z 330.683,A -85,B 0,C 180,E1 -11394.517,E2 -11394.517} C_VEL
LIN {X 0,Y 396.999,Z 333.299,A -85,B 0,C 180,E1 -11396.717,E2 -11396.717} C_VEL
LIN {X 0,Y 396.783,Z 337.573,A -85,B 0,C 180,E1 -11400.269,E2 -11400.269} C_VEL
LIN {X 0,Y 396.548,Z 341.855,A -85,B 0,C 180,E1 -11403.701,E2 -11403.701} C_VEL
LIN {X 0,Y 396.381,Z 346.425,A -85,B 0,C 180,E1 -11407.218,E2 -11407.218} C_VEL
LIN {X 0,Y 396.247,Z 350.603,A -85,B 0,C 180,E1 -11410.307,E2 -11410.307} C_VEL
LIN {X 0,Y 396.198,Z 352.733,A -85,B 0,C 180,E1 -11411.841,E2 -11411.841} C_VEL
LIN {X 0,Y 399.407,Z 366.161,A -85,B 0,C 180,E1 -11412.455,E2 -11412.455} C_VEL
LIN {X 0,Y 401.679,Z 377.63,A -85,B 0,C 180,E1 -11413.139,E2 -11413.139} C_VEL
LIN {X 0,Y 400.975,Z 390.387,A -85,B 0,C 180,E1 -11413.976,E2 -11413.976} C_VEL
LIN {X 0,Y 400.163,Z 401.104,A -85,B 0,C 180,E1 -11414.892,E2 -11414.892} C_VEL
LIN {X 0,Y 399.49,Z 411.427,A -85,B 0,C 180,E1 -11416.002,E2 -11416.002} C_VEL
LIN {X 0,Y 398.604,Z 421.036,A -85,B 0,C 180,E1 -11417.269,E2 -11417.269} C_VEL
LIN {X 0,Y 397.956,Z 428.902,A -85,B 0,C 180,E1 -11418.541,E2 -11418.541} C_VEL
LIN {X 0,Y 397.258,Z 436.591,A -85,B 0,C 180,E1 -11420.068,E2 -11420.068} C_VEL
LIN {X 0,Y 396.608,Z 443.647,A -85,B 0,C 180,E1 -11421.851,E2 -11421.851} C_VEL
LIN {X 0,Y 396.266,Z 448.158,A -85,B 0,C 180,E1 -11423.313,E2 -11423.313} C_VEL
LIN {X 0,Y 396.064,Z 451.94,A -85,B 0,C 180,E1 -11424.91,E2 -11424.91} C_VEL
LIN {X 0,Y 395.901,Z 453.8,A -85,B 0,C 180,E1 -11425.929,E2 -11425.929} C_VEL
LIN {X 0,Y 395.87,Z 455.198,A -85,B 0,C 180,E1 -11426.947,E2 -11426.947} C_VEL
LIN {X 0,Y 395.86,Z 456.191,A -85,B 0,C 180,E1 -11427.966,E2 -11427.966} C_VEL
LIN {X 0,Y 395.779,Z 457.038,A -85,B 0,C 180,E1 -11430,E2 -11430} C_VEL
LIN {X 0,Y 395.797,Z 456.849,A -85,B 0,C 180,E1 -11431.018,E2 -11431.018} C_VEL
LIN {X 0,Y 395.861,Z 456.264,A -85,B 0,C 180,E1 -11432.035,E2 -11432.035} C_VEL
LIN {X 0,Y 395.898,Z 453.945,A -85,B 0,C 180,E1 -11434.072,E2 -11434.072} C_VEL
LIN {X 0,Y 396.155,Z 451.079,A -85,B 0,C 180,E1 -11435.6,E2 -11435.6} C_VEL
LIN {X 0,Y 396.363,Z 447.197,A -85,B 0,C 180,E1 -11437.13,E2 -11437.13} C_VEL
LIN {X 0,Y 396.732,Z 442.186,A -85,B 0,C 180,E1 -11438.661,E2 -11438.661} C_VEL
LIN {X 0,Y 397.292,Z 435.875,A -85,B 0,C 180,E1 -11440.189,E2 -11440.189} C_VEL
LIN {X 0,Y 397.981,Z 427.975,A -85,B 0,C 180,E1 -11441.717,E2 -11441.717} C_VEL
LIN {X 0,Y 398.895,Z 418.144,A -85,B 0,C 180,E1 -11443.241,E2 -11443.241} C_VEL
LIN {X 0,Y 399.718,Z 408.454,A -85,B 0,C 180,E1 -11444.44,E2 -11444.44} C_VEL
LIN {X 0,Y 400.425,Z 397.716,A -85,B 0,C 180,E1 -11445.515,E2 -11445.515} C_VEL
LIN {X 0,Y 400.15,Z 392.707,A -85,B 0,C 180,E1 -11445.968,E2 -11445.968} C_VEL
LIN {X 0,Y 398.952,Z 387.748,A -85,B 0,C 180,E1 -11446.412,E2 -11446.412} C_VEL
LIN {X 0,Y 394.26,Z 374.335,A -85,B 0,C 180,E1 -11447.492,E2 -11447.492} C_VEL
LIN {X 0,Y 393.334,Z 370.758,A -85,B 0,C 180,E1 -11447.721,E2 -11447.721} C_VEL
LIN {X 0,Y 390.347,Z 358.006,A -85,B 0,C 180,E1 -11448.39,E2 -11448.39} C_VEL
LIN {X 0,Y 389.091,Z 352.917,A -85,B 0,C 180,E1 -11448.631,E2 -11448.631} C_VEL
LIN {X 0,Y 389.209,Z 349.452,A -85,B 0,C 180,E1 -11451.17,E2 -11451.17} C_VEL
LIN {X 0,Y 389.383,Z 345.079,A -85,B 0,C 180,E1 -11454.527,E2 -11454.527} C_VEL
LIN {X 0,Y 389.618,Z 340.737,A -85,B 0,C 180,E1 -11457.969,E2 -11457.969} C_VEL
LIN {X 0,Y 389.838,Z 336.42,A -85,B 0,C 180,E1 -11461.521,E2 -11461.521} C_VEL
LIN {X 0,Y 389.992,Z 333.456,A -85,B 0,C 180,E1 -11464.008,E2 -11464.008} C_VEL
LIN {X 0,Y 389.982,Z 331.408,A -85,B 0,C 180,E1 -11465.81,E2 -11465.81} C_VEL
LIN {X 0,Y 389.979,Z 330.913,A -85,B 0,C 180,E1 -11466.492,E2 -11466.492} C_VEL
LIN {X 0,Y 390.066,Z 330.898,A -85,B 0,C 180,E1 -11469.217,E2 -11469.217} C_VEL
LIN {X 0,Y 390.042,Z 330.897,A -85,B 0,C 180,E1 -11472.374,E2 -11472.374} C_VEL
LIN {X 0,Y 390.04,Z 330.901,A -85,B 0,C 180,E1 -11475.353,E2 -11475.353} C_VEL
LIN {X 0,Y 390.013,Z 330.901,A -85,B 0,C 180,E1 -11478.184,E2 -11478.184} C_VEL
LIN {X 0,Y 390.056,Z 330.897,A -85,B 0,C 180,E1 -11480.903,E2 -11480.903} C_VEL
LIN {X 0,Y 390.084,Z 330.893,A -85,B 0,C 180,E1 -11484.793,E2 -11484.793} C_VEL
LIN {X 0,Y 390.02,Z 330.9,A -85,B 0,C 180,E1 -11488.495,E2 -11488.495} C_VEL
LIN {X 0,Y 390.025,Z 330.899,A -85,B 0,C 180,E1 -11492.063,E2 -11492.063} C_VEL
LIN {X 0,Y 390.047,Z 330.898,A -85,B 0,C 180,E1 -11495.517,E2 -11495.517} C_VEL
LIN {X 0,Y 390.052,Z 330.901,A -85,B 0,C 180,E1 -11498.877,E2 -11498.877} C_VEL
LIN {X 0,Y 390.125,Z 330.887,A -85,B 0,C 180,E1 -11502.166,E2 -11502.166} C_VEL
LIN {X 0,Y 390.139,Z 330.885,A -85,B 0,C 180,E1 -11505.392,E2 -11505.392} C_VEL
LIN {X 0,Y 390.144,Z 330.89,A -85,B 0,C 180,E1 -11508.571,E2 -11508.571} C_VEL
LIN {X 0,Y 390.341,Z 330.861,A -85,B 0,C 180,E1 -11511.993,E2 -11511.993} C_VEL
LIN {X 0,Y 390.224,Z 330.877,A -85,B 0,C 180,E1 -11514.833,E2 -11514.833} C_VEL
LIN {X 0,Y 390.413,Z 330.852,A -85,B 0,C 180,E1 -11517.937,E2 -11517.937} C_VEL
LIN {X 0,Y 390.534,Z 330.838,A -85,B 0,C 180,E1 -11520,E2 -11520} C_VEL
LIN {X 0,Y 390.305,Z 330.864,A -85,B 0,C 180,E1 -11523.097,E2 -11523.097} C_VEL
LIN {X 0,Y 390.324,Z 330.867,A -85,B 0,C 180,E1 -11526.202,E2 -11526.202} C_VEL
LIN {X 0,Y 390.201,Z 330.877,A -85,B 0,C 180,E1 -11529.329,E2 -11529.329} C_VEL
LIN {X 0,Y 390.191,Z 330.879,A -85,B 0,C 180,E1 -11533.439,E2 -11533.439} C_VEL
LIN {X 0,Y 390.145,Z 330.885,A -85,B 0,C 180,E1 -11537.308,E2 -11537.308} C_VEL
LIN {X 0,Y 390.084,Z 330.892,A -85,B 0,C 180,E1 -11540.47,E2 -11540.47} C_VEL
LIN {X 0,Y 390.071,Z 330.896,A -85,B 0,C 180,E1 -11543.352,E2 -11543.352} C_VEL
LIN {X 0,Y 390.045,Z 330.896,A -85,B 0,C 180,E1 -11546.773,E2 -11546.773} C_VEL
LIN {X 0,Y 390.034,Z 330.898,A -85,B 0,C 180,E1 -11550.3,E2 -11550.3} C_VEL
LIN {X 0,Y 390.066,Z 330.895,A -85,B 0,C 180,E1 -11554.025,E2 -11554.025} C_VEL
LIN {X 0,Y 390.04,Z 330.901,A -85,B 0,C 180,E1 -11557.551,E2 -11557.551} C_VEL
LIN {X 0,Y 390.014,Z 330.902,A -85,B 0,C 180,E1 -11560.815,E2 -11560.815} C_VEL
LIN {X 0,Y 390.042,Z 330.899,A -85,B 0,C 180,E1 -11563.885,E2 -11563.885} C_VEL
LIN {X 0,Y 390.059,Z 330.9,A -85,B 0,C 180,E1 -11566.79,E2 -11566.79} C_VEL
LIN {X 0,Y 390.071,Z 330.975,A -85,B 0,C 180,E1 -11567.91,E2 -11567.91} C_VEL
LIN {X 0,Y 390.938,Z 335.817,A -85,B 0,C 180,E1 -11571.009,E2 -11571.009} C_VEL
LIN {X 0,Y 391.426,Z 340.235,A -85,B 0,C 180,E1 -11573.665,E2 -11573.665} C_VEL
LIN {X 0,Y 391.407,Z 343.786,A -85,B 0,C 180,E1 -11575.686,E2 -11575.686} C_VEL
LIN {X 0,Y 390.917,Z 350.195,A -85,B 0,C 180,E1 -11579.178,E2 -11579.178} C_VEL
LIN {X 0,Y 390.388,Z 356.871,A -85,B 0,C 180,E1 -11582.673,E2 -11582.673} C_VEL
LIN {X 0,Y 389.955,Z 363.479,A -85,B 0,C 180,E1 -11586.077,E2 -11586.077} C_VEL
LIN {X 0,Y 389.564,Z 371.131,A -85,B 0,C 180,E1 -11589.954,E2 -11589.954} C_VEL
LIN {X 0,Y 389.412,Z 374.184,A -85,B 0,C 180,E1 -11591.436,E2 -11591.436} C_VEL
LIN {X 0,Y 391.95,Z 387.512,A -85,B 0,C 180,E1 -11591.991,E2 -11591.991} C_VEL
LIN {X 0,Y 393.991,Z 401.026,A -85,B 0,C 180,E1 -11592.767,E2 -11592.767} C_VEL
LIN {X 0,Y 394.278,Z 406.138,A -85,B 0,C 180,E1 -11593.105,E2 -11593.105} C_VEL
LIN {X 0,Y 393.441,Z 417.313,A -85,B 0,C 180,E1 -11593.926,E2 -11593.926} C_VEL
LIN {X 0,Y 392.52,Z 428.774,A -85,B 0,C 180,E1 -11595.005,E2 -11595.005} C_VEL
LIN {X 0,Y 391.624,Z 439.256,A -85,B 0,C 180,E1 -11596.252,E2 -11596.252} C_VEL
LIN {X 0,Y 390.857,Z 448.047,A -85,B 0,C 180,E1 -11597.539,E2 -11597.539} C_VEL
LIN {X 0,Y 390.079,Z 456.68,A -85,B 0,C 180,E1 -11599.095,E2 -11599.095} C_VEL
LIN {X 0,Y 389.503,Z 463.583,A -85,B 0,C 180,E1 -11600.654,E2 -11600.654} C_VEL
LIN {X 0,Y 389.094,Z 469.117,A -85,B 0,C 180,E1 -11602.214,E2 -11602.214} C_VEL
LIN {X 0,Y 388.854,Z 473.459,A -85,B 0,C 180,E1 -11603.774,E2 -11603.774} C_VEL
LIN {X 0,Y 388.782,Z 475.759,A -85,B 0,C 180,E1 -11604.814,E2 -11604.814} C_VEL
LIN {X 0,Y 388.715,Z 477.624,A -85,B 0,C 180,E1 -11605.852,E2 -11605.852} C_VEL
LIN {X 0,Y 388.659,Z 480.02,A -85,B 0,C 180,E1 -11607.927,E2 -11607.927} C_VEL
LIN {X 0,Y 388.689,Z 480.63,A -85,B 0,C 180,E1 -11608.964,E2 -11608.964} C_VEL
LIN {X 0,Y 388.675,Z 480.847,A -85,B 0,C 180,E1 -11610,E2 -11610} C_VEL
LIN {X 0,Y 388.689,Z 480.631,A -85,B 0,C 180,E1 -11611.036,E2 -11611.036} C_VEL
LIN {X 0,Y 388.659,Z 480.021,A -85,B 0,C 180,E1 -11612.072,E2 -11612.072} C_VEL
LIN {X 0,Y 388.715,Z 477.627,A -85,B 0,C 180,E1 -11614.147,E2 -11614.147} C_VEL
LIN {X 0,Y 388.796,Z 474.351,A -85,B 0,C 180,E1 -11615.854,E2 -11615.854} C_VEL
LIN {X 0,Y 389.094,Z 469.114,A -85,B 0,C 180,E1 -11617.785,E2 -11617.785} C_VEL
LIN {X 0,Y 389.514,Z 463.582,A -85,B 0,C 180,E1 -11619.345,E2 -11619.345} C_VEL
LIN {X 0,Y 390.078,Z 456.677,A -85,B 0,C 180,E1 -11620.904,E2 -11620.904} C_VEL
LIN {X 0,Y 390.869,Z 448.042,A -85,B 0,C 180,E1 -11622.46,E2 -11622.46} C_VEL
LIN {X 0,Y 391.69,Z 439.267,A -85,B 0,C 180,E1 -11623.742,E2 -11623.742} C_VEL
LIN {X 0,Y 392.507,Z 428.764,A -85,B 0,C 180,E1 -11624.994,E2 -11624.994} C_VEL
LIN {X 0,Y 393.313,Z 418.841,A -85,B 0,C 180,E1 -11625.945,E2 -11625.945} C_VEL
LIN {X 0,Y 394.216,Z 407.729,A -85,B 0,C 180,E1 -11626.789,E2 -11626.789} C_VEL
LIN {X 0,Y 394.196,Z 402.83,A -85,B 0,C 180,E1 -11627.115,E2 -11627.115} C_VEL
LIN {X 0,Y 392.294,Z 389.907,A -85,B 0,C 180,E1 -11627.884,E2 -11627.884} C_VEL
LIN {X 0,Y 389.851,Z 376.424,A -85,B 0,C 180,E1 -11628.484,E2 -11628.484} C_VEL
LIN {X 0,Y 389.405,Z 374.028,A -85,B 0,C 180,E1 -11628.581,E2 -11628.581} C_VEL
LIN {X 0,Y 389.76,Z 366.778,A -85,B 0,C 180,E1 -11632.25,E2 -11632.25} C_VEL
LIN {X 0,Y 390.185,Z 359.891,A -85,B 0,C 180,E1 -11635.763,E2 -11635.763} C_VEL
LIN {X 0,Y 390.603,Z 353.516,A -85,B 0,C 180,E1 -11639.064,E2 -11639.064} C_VEL
LIN {X 0,Y 390.963,Z 349.065,A -85,B 0,C 180,E1 -11641.419,E2 -11641.419} C_VEL
LIN {X 0,Y 391.404,Z 343.75,A -85,B 0,C 180,E1 -11644.313,E2 -11644.313} C_VEL
LIN {X 0,Y 391.377,Z 339.109,A -85,B 0,C 180,E1 -11646.98,E2 -11646.98} C_VEL
LIN {X 0,Y 390.879,Z 335.194,A -85,B 0,C 180,E1 -11649.363,E2 -11649.363} C_VEL
LIN {X 0,Y 390.139,Z 330.891,A -85,B 0,C 180,E1 -11652.194,E2 -11652.194} C_VEL
LIN {X 0,Y 390.056,Z 330.903,A -85,B 0,C 180,E1 -11655.356,E2 -11655.356} C_VEL
LIN {X 0,Y 390.011,Z 330.901,A -85,B 0,C 180,E1 -11658.184,E2 -11658.184} C_VEL
LIN {X 0,Y 390.057,Z 330.899,A -85,B 0,C 180,E1 -11660.904,E2 -11660.904} C_VEL
LIN {X 0,Y 390.079,Z 330.897,A -85,B 0,C 180,E1 -11664.792,E2 -11664.792} C_VEL
LIN {X 0,Y 390.015,Z 330.905,A -85,B 0,C 180,E1 -11668.495,E2 -11668.495} C_VEL
LIN {X 0,Y 390.021,Z 330.902,A -85,B 0,C 180,E1 -11672.062,E2 -11672.062} C_VEL
LIN {X 0,Y 390.047,Z 330.896,A -85,B 0,C 180,E1 -11675.517,E2 -11675.517} C_VEL
LIN {X 0,Y 390.047,Z 330.897,A -85,B 0,C 180,E1 -11678.877,E2 -11678.877} C_VEL
LIN {X 0,Y 390.119,Z 330.892,A -85,B 0,C 180,E1 -11682.166,E2 -11682.166} C_VEL
LIN {X 0,Y 390.133,Z 330.886,A -85,B 0,C 180,E1 -11685.392,E2 -11685.392} C_VEL
LIN {X 0,Y 390.138,Z 330.886,A -85,B 0,C 180,E1 -11688.571,E2 -11688.571} C_VEL
LIN {X 0,Y 390.334,Z 330.865,A -85,B 0,C 180,E1 -11691.993,E2 -11691.993} C_VEL
LIN {X 0,Y 390.225,Z 330.874,A -85,B 0,C 180,E1 -11694.834,E2 -11694.834} C_VEL
LIN {X 0,Y 390.41,Z 330.856,A -85,B 0,C 180,E1 -11697.937,E2 -11697.937} C_VEL
LIN {X 0,Y 390.531,Z 330.839,A -85,B 0,C 180,E1 -11700,E2 -11700} C_VEL
LIN {X 0,Y 390.302,Z 330.866,A -85,B 0,C 180,E1 -11703.097,E2 -11703.097} C_VEL
LIN {X 0,Y 390.302,Z 330.865,A -85,B 0,C 180,E1 -11706.591,E2 -11706.591} C_VEL
LIN {X 0,Y 390.195,Z 330.883,A -85,B 0,C 180,E1 -11709.329,E2 -11709.329} C_VEL
LIN {X 0,Y 390.185,Z 330.884,A -85,B 0,C 180,E1 -11713.439,E2 -11713.439} C_VEL
LIN {X 0,Y 390.14,Z 330.89,A -85,B 0,C 180,E1 -11717.308,E2 -11717.308} C_VEL
LIN {X 0,Y 390.079,Z 330.893,A -85,B 0,C 180,E1 -11720.471,E2 -11720.471} C_VEL
LIN {X 0,Y 390.066,Z 330.898,A -85,B 0,C 180,E1 -11723.353,E2 -11723.353} C_VEL
LIN {X 0,Y 390.04,Z 330.902,A -85,B 0,C 180,E1 -11726.774,E2 -11726.774} C_VEL
LIN {X 0,Y 390.029,Z 330.899,A -85,B 0,C 180,E1 -11730.301,E2 -11730.301} C_VEL
LIN {X 0,Y 390.061,Z 330.895,A -85,B 0,C 180,E1 -11734.025,E2 -11734.025} C_VEL
LIN {X 0,Y 390.033,Z 330.898,A -85,B 0,C 180,E1 -11737.551,E2 -11737.551} C_VEL
LIN {X 0,Y 390.01,Z 330.905,A -85,B 0,C 180,E1 -11740.816,E2 -11740.816} C_VEL
LIN {X 0,Y 390.046,Z 330.897,A -85,B 0,C 180,E1 -11743.887,E2 -11743.887} C_VEL
LIN {X 0,Y 390.076,Z 330.893,A -85,B 0,C 180,E1 -11747.621,E2 -11747.621} C_VEL
LIN {X 0,Y 390.09,Z 330.892,A -85,B 0,C 180,E1 -11750.909,E2 -11750.909} C_VEL
LIN {X 0,Y 389.973,Z 330.912,A -85,B 0,C 180,E1 -11753.509,E2 -11753.509} C_VEL
LIN {X 0,Y 389.996,Z 331.958,A -85,B 0,C 180,E1 -11754.785,E2 -11754.785} C_VEL
LIN {X 0,Y 389.879,Z 335.655,A -85,B 0,C 180,E1 -11757.912,E2 -11757.912} C_VEL
LIN {X 0,Y 389.672,Z 339.169,A -85,B 0,C 180,E1 -11760.86,E2 -11760.86} C_VEL
LIN {X 0,Y 389.487,Z 343.621,A -85,B 0,C 180,E1 -11764.451,E2 -11764.451} C_VEL
LIN {X 0,Y 389.283,Z 347.85,A -85,B 0,C 180,E1 -11767.721,E2 -11767.721} C_VEL
LIN {X 0,Y 389.127,Z 352.311,A -85,B 0,C 180,E1 -11771.029,E2 -11771.029} C_VEL
LIN {X 0,Y 389.142,Z 353.005,A -85,B 0,C 180,E1 -11771.501,E2 -11771.501} C_VEL
LIN {X 0,Y 392.328,Z 366.086,A -85,B 0,C 180,E1 -11772.114,E2 -11772.114} C_VEL
LIN {X 0,Y 394.801,Z 378.44,A -85,B 0,C 180,E1 -11772.871,E2 -11772.871} C_VEL
LIN {X 0,Y 394.166,Z 390.609,A -85,B 0,C 180,E1 -11773.691,E2 -11773.691} C_VEL
LIN {X 0,Y 393.302,Z 401.66,A -85,B 0,C 180,E1 -11774.657,E2 -11774.657} C_VEL
LIN {X 0,Y 392.511,Z 412.711,A -85,B 0,C 180,E1 -11775.88,E2 -11775.88} C_VEL
LIN {X 0,Y 391.678,Z 421.255,A -85,B 0,C 180,E1 -11777.04,E2 -11777.04} C_VEL
LIN {X 0,Y 391.004,Z 429.12,A -85,B 0,C 180,E1 -11778.334,E2 -11778.334} C_VEL
LIN {X 0,Y 390.251,Z 436.809,A -85,B 0,C 180,E1 -11779.888,E2 -11779.888} C_VEL
LIN {X 0,Y 389.559,Z 443.865,A -85,B 0,C 180,E1 -11781.702,E2 -11781.702} C_VEL
LIN {X 0,Y 389.196,Z 448.686,A -85,B 0,C 180,E1 -11783.305,E2 -11783.305} C_VEL
LIN {X 0,Y 389.012,Z 452.156,A -85,B 0,C 180,E1 -11784.818,E2 -11784.818} C_VEL
LIN {X 0,Y 388.826,Z 454.016,A -85,B 0,C 180,E1 -11785.854,E2 -11785.854} C_VEL
LIN {X 0,Y 388.775,Z 455.414,A -85,B 0,C 180,E1 -11786.892,E2 -11786.892} C_VEL
LIN {X 0,Y 388.763,Z 456.407,A -85,B 0,C 180,E1 -11787.928,E2 -11787.928} C_VEL
LIN {X 0,Y 388.708,Z 457.253,A -85,B 0,C 180,E1 -11790,E2 -11790} C_VEL
LIN {X 0,Y 388.729,Z 457.063,A -85,B 0,C 180,E1 -11791.036,E2 -11791.036} C_VEL
LIN {X 0,Y 388.763,Z 456.479,A -85,B 0,C 180,E1 -11792.072,E2 -11792.072} C_VEL
LIN {X 0,Y 388.823,Z 454.16,A -85,B 0,C 180,E1 -11794.146,E2 -11794.146} C_VEL
LIN {X 0,Y 389.088,Z 451.293,A -85,B 0,C 180,E1 -11795.702,E2 -11795.702} C_VEL
LIN {X 0,Y 389.314,Z 447.411,A -85,B 0,C 180,E1 -11797.26,E2 -11797.26} C_VEL
LIN {X 0,Y 389.704,Z 442.4,A -85,B 0,C 180,E1 -11798.818,E2 -11798.818} C_VEL
LIN {X 0,Y 390.299,Z 436.088,A -85,B 0,C 180,E1 -11800.374,E2 -11800.374} C_VEL
LIN {X 0,Y 391.024,Z 428.188,A -85,B 0,C 180,E1 -11801.929,E2 -11801.929} C_VEL
LIN {X 0,Y 391.812,Z 420.131,A -85,B 0,C 180,E1 -11803.221,E2 -11803.221} C_VEL
LIN {X 0,Y 392.734,Z 410.297,A -85,B 0,C 180,E1 -11804.509,E2 -11804.509} C_VEL
LIN {X 0,Y 393.411,Z 400.624,A -85,B 0,C 180,E1 -11805.543,E2 -11805.543} C_VEL
LIN {X 0,Y 394.211,Z 390.15,A -85,B 0,C 180,E1 -11806.441,E2 -11806.441} C_VEL
LIN {X 0,Y 394.888,Z 379.202,A -85,B 0,C 180,E1 -11807.178,E2 -11807.178} C_VEL
LIN {X 0,Y 393.334,Z 370.758,A -85,B 0,C 180,E1 -11807.721,E2 -11807.721} C_VEL
LIN {X 0,Y 391.941,Z 367.391,A -85,B 0,C 180,E1 -11807.955,E2 -11807.955} C_VEL
LIN {X 0,Y 387.924,Z 362.673,A -85,B 0,C 180,E1 -11808.353,E2 -11808.353} C_VEL
LIN {X 0,Y 383.815,Z 357.898,A -85,B 0,C 180,E1 -11808.724,E2 -11808.724} C_VEL
LIN {X 0,Y 382.265,Z 354.434,A -85,B 0,C 180,E1 -11808.91,E2 -11808.91} C_VEL
LIN {X 0,Y 382.04,Z 353.128,A -85,B 0,C 180,E1 -11808.988,E2 -11808.988} C_VEL
LIN {X 0,Y 382.153,Z 349.654,A -85,B 0,C 180,E1 -11811.581,E2 -11811.581} C_VEL
LIN {X 0,Y 382.353,Z 345.27,A -85,B 0,C 180,E1 -11815.009,E2 -11815.009} C_VEL
LIN {X 0,Y 382.6,Z 340.911,A -85,B 0,C 180,E1 -11818.528,E2 -11818.528} C_VEL
LIN {X 0,Y 382.872,Z 336.56,A -85,B 0,C 180,E1 -11822.162,E2 -11822.162} C_VEL
LIN {X 0,Y 382.956,Z 333.685,A -85,B 0,C 180,E1 -11824.674,E2 -11824.674} C_VEL
LIN {X 0,Y 382.938,Z 332.025,A -85,B 0,C 180,E1 -11826.145,E2 -11826.145} C_VEL
LIN {X 0,Y 382.999,Z 331.779,A -85,B 0,C 180,E1 -11828.601,E2 -11828.601} C_VEL
LIN {X 0,Y 382.984,Z 331.779,A -85,B 0,C 180,E1 -11831.347,E2 -11831.347} C_VEL
LIN {X 0,Y 382.995,Z 331.775,A -85,B 0,C 180,E1 -11834.303,E2 -11834.303} C_VEL
LIN {X 0,Y 382.98,Z 331.78,A -85,B 0,C 180,E1 -11837.236,E2 -11837.236} C_VEL
LIN {X 0,Y 382.984,Z 331.776,A -85,B 0,C 180,E1 -11840.419,E2 -11840.419} C_VEL
LIN {X 0,Y 383.023,Z 331.772,A -85,B 0,C 180,E1 -11844.044,E2 -11844.044} C_VEL
LIN {X 0,Y 382.984,Z 331.779,A -85,B 0,C 180,E1 -11847.578,E2 -11847.578} C_VEL
LIN {X 0,Y 382.975,Z 331.777,A -85,B 0,C 180,E1 -11850.298,E2 -11850.298} C_VEL
LIN {X 0,Y 383.001,Z 331.774,A -85,B 0,C 180,E1 -11854.044,E2 -11854.044} C_VEL
LIN {X 0,Y 382.989,Z 331.778,A -85,B 0,C 180,E1 -11857.334,E2 -11857.334} C_VEL
LIN {X 0,Y 383.057,Z 331.772,A -85,B 0,C 180,E1 -11860.716,E2 -11860.716} C_VEL
LIN {X 0,Y 383.076,Z 331.764,A -85,B 0,C 180,E1 -11864.026,E2 -11864.026} C_VEL
LIN {X 0,Y 383.133,Z 331.759,A -85,B 0,C 180,E1 -11867.284,E2 -11867.284} C_VEL
LIN {X 0,Y 383.148,Z 331.761,A -85,B 0,C 180,E1 -11870.498,E2 -11870.498} C_VEL
LIN {X 0,Y 383.27,Z 331.746,A -85,B 0,C 180,E1 -11872.625,E2 -11872.625} C_VEL
LIN {X 0,Y 383.196,Z 331.753,A -85,B 0,C 180,E1 -11874.738,E2 -11874.738} C_VEL
LIN {X 0,Y 383.381,Z 331.728,A -85,B 0,C 180,E1 -11877.899,E2 -11877.899} C_VEL
LIN {X 0,Y 383.504,Z 331.714,A -85,B 0,C 180,E1 -11880,E2 -11880} C_VEL
LIN {X 0,Y 383.242,Z 331.744,A -85,B 0,C 180,E1 -11883.154,E2 -11883.154} C_VEL
LIN {X 0,Y 383.28,Z 331.744,A -85,B 0,C 180,E1 -11886.316,E2 -11886.316} C_VEL
LIN {X 0,Y 383.148,Z 331.757,A -85,B 0,C 180,E1 -11889.502,E2 -11889.502} C_VEL
LIN {X 0,Y 383.122,Z 331.76,A -85,B 0,C 180,E1 -11893.536,E2 -11893.536} C_VEL
LIN {X 0,Y 383.091,Z 331.765,A -85,B 0,C 180,E1 -11897.455,E2 -11897.455} C_VEL
LIN {X 0,Y 383.025,Z 331.771,A -85,B 0,C 180,E1 -11900.647,E2 -11900.647} C_VEL
LIN {X 0,Y 383.016,Z 331.777,A -85,B 0,C 180,E1 -11903.808,E2 -11903.808} C_VEL
LIN {X 0,Y 382.983,Z 331.779,A -85,B 0,C 180,E1 -11907.308,E2 -11907.308} C_VEL
LIN {X 0,Y 382.979,Z 331.778,A -85,B 0,C 180,E1 -11910.919,E2 -11910.919} C_VEL
LIN {X 0,Y 383.016,Z 331.772,A -85,B 0,C 180,E1 -11914.668,E2 -11914.668} C_VEL
LIN {X 0,Y 382.993,Z 331.776,A -85,B 0,C 180,E1 -11917.903,E2 -11917.903} C_VEL
LIN {X 0,Y 382.958,Z 331.784,A -85,B 0,C 180,E1 -11921.351,E2 -11921.351} C_VEL
LIN {X 0,Y 382.988,Z 331.779,A -85,B 0,C 180,E1 -11924.303,E2 -11924.303} C_VEL
LIN {X 0,Y 383.017,Z 331.85,A -85,B 0,C 180,E1 -11927.598,E2 -11927.598} C_VEL
LIN {X 0,Y 383.755,Z 335.924,A -85,B 0,C 180,E1 -11930.28,E2 -11930.28} C_VEL
LIN {X 0,Y 384.358,Z 340.104,A -85,B 0,C 180,E1 -11932.886,E2 -11932.886} C_VEL
LIN {X 0,Y 384.424,Z 344.517,A -85,B 0,C 180,E1 -11935.477,E2 -11935.477} C_VEL
LIN {X 0,Y 383.941,Z 350.039,A -85,B 0,C 180,E1 -11938.555,E2 -11938.555} C_VEL
LIN {X 0,Y 383.472,Z 355.711,A -85,B 0,C 180,E1 -11941.608,E2 -11941.608} C_VEL
LIN {X 0,Y 383.021,Z 362.203,A -85,B 0,C 180,E1 -11945.038,E2 -11945.038} C_VEL
LIN {X 0,Y 382.588,Z 369.856,A -85,B 0,C 180,E1 -11949.01,E2 -11949.01} C_VEL
LIN {X 0,Y 382.363,Z 373.975,A -85,B 0,C 180,E1 -11951.081,E2 -11951.081} C_VEL
LIN {X 0,Y 384.905,Z 387.108,A -85,B 0,C 180,E1 -11951.642,E2 -11951.642} C_VEL
LIN {X 0,Y 386.769,Z 399.599,A -85,B 0,C 180,E1 -11952.362,E2 -11952.362} C_VEL
LIN {X 0,Y 387.47,Z 406.166,A -85,B 0,C 180,E1 -11952.815,E2 -11952.815} C_VEL
LIN {X 0,Y 386.489,Z 418.64,A -85,B 0,C 180,E1 -11953.765,E2 -11953.765} C_VEL
LIN {X 0,Y 385.493,Z 430.45,A -85,B 0,C 180,E1 -11954.942,E2 -11954.942} C_VEL
LIN {X 0,Y 384.527,Z 440.931,A -85,B 0,C 180,E1 -11956.255,E2 -11956.255} C_VEL
LIN {X 0,Y 383.745,Z 449.419,A -85,B 0,C 180,E1 -11957.573,E2 -11957.573} C_VEL
LIN {X 0,Y 382.978,Z 457.703,A -85,B 0,C 180,E1 -11959.158,E2 -11959.158} C_VEL
LIN {X 0,Y 382.41,Z 464.382,A -85,B 0,C 180,E1 -11960.746,E2 -11960.746} C_VEL
LIN {X 0,Y 381.96,Z 470.497,A -85,B 0,C 180,E1 -11962.599,E2 -11962.599} C_VEL
LIN {X 0,Y 381.749,Z 473.568,A -85,B 0,C 180,E1 -11963.795,E2 -11963.795} C_VEL
LIN {X 0,Y 381.642,Z 477.409,A -85,B 0,C 180,E1 -11965.775,E2 -11965.775} C_VEL
LIN {X 0,Y 381.558,Z 479.804,A -85,B 0,C 180,E1 -11967.888,E2 -11967.888} C_VEL
LIN {X 0,Y 381.59,Z 480.415,A -85,B 0,C 180,E1 -11968.944,E2 -11968.944} C_VEL
LIN {X 0,Y 381.59,Z 480.632,A -85,B 0,C 180,E1 -11970,E2 -11970} C_VEL
LIN {X 0,Y 381.59,Z 480.415,A -85,B 0,C 180,E1 -11971.055,E2 -11971.055} C_VEL
LIN {X 0,Y 381.558,Z 479.806,A -85,B 0,C 180,E1 -11972.111,E2 -11972.111} C_VEL
LIN {X 0,Y 381.641,Z 477.411,A -85,B 0,C 180,E1 -11974.224,E2 -11974.224} C_VEL
LIN {X 0,Y 381.748,Z 473.566,A -85,B 0,C 180,E1 -11976.203,E2 -11976.203} C_VEL
LIN {X 0,Y 382.052,Z 468.897,A -85,B 0,C 180,E1 -11977.93,E2 -11977.93} C_VEL
LIN {X 0,Y 382.477,Z 463.364,A -85,B 0,C 180,E1 -11979.518,E2 -11979.518} C_VEL
LIN {X 0,Y 383.05,Z 456.458,A -85,B 0,C 180,E1 -11981.107,E2 -11981.107} C_VEL
LIN {X 0,Y 383.919,Z 447.824,A -85,B 0,C 180,E1 -11982.689,E2 -11982.689} C_VEL
LIN {X 0,Y 384.725,Z 439.235,A -85,B 0,C 180,E1 -11983.97,E2 -11983.97} C_VEL
LIN {X 0,Y 385.571,Z 429.251,A -85,B 0,C 180,E1 -11985.189,E2 -11985.189} C_VEL
LIN {X 0,Y 386.467,Z 418.622,A -85,B 0,C 180,E1 -11986.235,E2 -11986.235} C_VEL
LIN {X 0,Y 387.444,Z 406.128,A -85,B 0,C 180,E1 -11987.185,E2 -11987.185} C_VEL
LIN {X 0,Y 386.032,Z 394.224,A -85,B 0,C 180,E1 -11987.965,E2 -11987.965} C_VEL
LIN {X 0,Y 383.84,Z 381.475,A -85,B 0,C 180,E1 -11988.622,E2 -11988.622} C_VEL
LIN {X 0,Y 382.336,Z 373.817,A -85,B 0,C 180,E1 -11988.938,E2 -11988.938} C_VEL
LIN {X 0,Y 382.683,Z 367.681,A -85,B 0,C 180,E1 -11992.115,E2 -11992.115} C_VEL
LIN {X 0,Y 383.02,Z 362.207,A -85,B 0,C 180,E1 -11994.961,E2 -11994.961} C_VEL
LIN {X 0,Y 383.475,Z 355.574,A -85,B 0,C 180,E1 -11998.456,E2 -11998.456} C_VEL
LIN {X 0,Y 383.936,Z 350.025,A -85,B 0,C 180,E1 -12001.445,E2 -12001.445} C_VEL
LIN {X 0,Y 384.42,Z 344.267,A -85,B 0,C 180,E1 -12004.644,E2 -12004.644} C_VEL
LIN {X 0,Y 384.357,Z 340.075,A -85,B 0,C 180,E1 -12007.113,E2 -12007.113} C_VEL
LIN {X 0,Y 383.75,Z 335.679,A -85,B 0,C 180,E1 -12009.864,E2 -12009.864} C_VEL
LIN {X 0,Y 383.096,Z 331.768,A -85,B 0,C 180,E1 -12012.479,E2 -12012.479} C_VEL
LIN {X 0,Y 383,Z 331.779,A -85,B 0,C 180,E1 -12015.789,E2 -12015.789} C_VEL
LIN {X 0,Y 382.956,Z 331.786,A -85,B 0,C 180,E1 -12018.799,E2 -12018.799} C_VEL
LIN {X 0,Y 382.99,Z 331.776,A -85,B 0,C 180,E1 -12022.096,E2 -12022.096} C_VEL
LIN {X 0,Y 383.011,Z 331.773,A -85,B 0,C 180,E1 -12025.331,E2 -12025.331} C_VEL
LIN {X 0,Y 382.974,Z 331.778,A -85,B 0,C 180,E1 -12029.081,E2 -12029.081} C_VEL
LIN {X 0,Y 382.978,Z 331.78,A -85,B 0,C 180,E1 -12032.692,E2 -12032.692} C_VEL
LIN {X 0,Y 383.01,Z 331.777,A -85,B 0,C 180,E1 -12036.191,E2 -12036.191} C_VEL
LIN {X 0,Y 383.046,Z 331.769,A -85,B 0,C 180,E1 -12039.598,E2 -12039.598} C_VEL
LIN {X 0,Y 383.096,Z 331.762,A -85,B 0,C 180,E1 -12042.931,E2 -12042.931} C_VEL
LIN {X 0,Y 383.116,Z 331.762,A -85,B 0,C 180,E1 -12046.464,E2 -12046.464} C_VEL
LIN {X 0,Y 383.142,Z 331.758,A -85,B 0,C 180,E1 -12050.498,E2 -12050.498} C_VEL
LIN {X 0,Y 383.264,Z 331.741,A -85,B 0,C 180,E1 -12052.625,E2 -12052.625} C_VEL
LIN {X 0,Y 383.197,Z 331.75,A -85,B 0,C 180,E1 -12054.738,E2 -12054.738} C_VEL
LIN {X 0,Y 383.377,Z 331.732,A -85,B 0,C 180,E1 -12057.899,E2 -12057.899} C_VEL
LIN {X 0,Y 383.5,Z 331.715,A -85,B 0,C 180,E1 -12060,E2 -12060} C_VEL
LIN {X 0,Y 383.239,Z 331.746,A -85,B 0,C 180,E1 -12063.154,E2 -12063.154} C_VEL
LIN {X 0,Y 383.263,Z 331.741,A -85,B 0,C 180,E1 -12066.584,E2 -12066.584} C_VEL
LIN {X 0,Y 383.251,Z 331.743,A -85,B 0,C 180,E1 -12068.436,E2 -12068.436} C_VEL
LIN {X 0,Y 383.088,Z 331.767,A -85,B 0,C 180,E1 -12071.642,E2 -12071.642} C_VEL
LIN {X 0,Y 383.099,Z 331.764,A -85,B 0,C 180,E1 -12074.882,E2 -12074.882} C_VEL
LIN {X 0,Y 383.054,Z 331.767,A -85,B 0,C 180,E1 -12078.174,E2 -12078.174} C_VEL
LIN {X 0,Y 382.984,Z 331.778,A -85,B 0,C 180,E1 -12081.532,E2 -12081.532} C_VEL
LIN {X 0,Y 383.01,Z 331.778,A -85,B 0,C 180,E1 -12084.963,E2 -12084.963} C_VEL
LIN {X 0,Y 382.973,Z 331.779,A -85,B 0,C 180,E1 -12088.498,E2 -12088.498} C_VEL
LIN {X 0,Y 383.001,Z 331.774,A -85,B 0,C 180,E1 -12092.151,E2 -12092.151} C_VEL
LIN {X 0,Y 383.011,Z 331.778,A -85,B 0,C 180,E1 -12094.669,E2 -12094.669} C_VEL
LIN {X 0,Y 382.987,Z 331.776,A -85,B 0,C 180,E1 -12097.903,E2 -12097.903} C_VEL
LIN {X 0,Y 382.955,Z 331.78,A -85,B 0,C 180,E1 -12101.352,E2 -12101.352} C_VEL
LIN {X 0,Y 382.989,Z 331.779,A -85,B 0,C 180,E1 -12104.304,E2 -12104.304} C_VEL
LIN {X 0,Y 383.035,Z 331.77,A -85,B 0,C 180,E1 -12107.245,E2 -12107.245} C_VEL
LIN {X 0,Y 383.017,Z 331.777,A -85,B 0,C 180,E1 -12110.414,E2 -12110.414} C_VEL
LIN {X 0,Y 382.968,Z 331.784,A -85,B 0,C 180,E1 -12112.73,E2 -12112.73} C_VEL
LIN {X 0,Y 382.943,Z 332.102,A -85,B 0,C 180,E1 -12114.037,E2 -12114.037} C_VEL
LIN {X 0,Y 382.918,Z 334.998,A -85,B 0,C 180,E1 -12116.592,E2 -12116.592} C_VEL
LIN {X 0,Y 382.667,Z 339.352,A -85,B 0,C 180,E1 -12120.274,E2 -12120.274} C_VEL
LIN {X 0,Y 382.454,Z 343.665,A -85,B 0,C 180,E1 -12123.832,E2 -12123.832} C_VEL
LIN {X 0,Y 382.268,Z 348.049,A -85,B 0,C 180,E1 -12127.29,E2 -12127.29} C_VEL
LIN {X 0,Y 382.089,Z 352.525,A -85,B 0,C 180,E1 -12130.666,E2 -12130.666} C_VEL
LIN {X 0,Y 382.084,Z 353.32,A -85,B 0,C 180,E1 -12131.149,E2 -12131.149} C_VEL
LIN {X 0,Y 385.366,Z 366.499,A -85,B 0,C 180,E1 -12131.788,E2 -12131.788} C_VEL
LIN {X 0,Y 387.654,Z 377.663,A -85,B 0,C 180,E1 -12132.484,E2 -12132.484} C_VEL
LIN {X 0,Y 387.957,Z 382.078,A -85,B 0,C 180,E1 -12132.779,E2 -12132.779} C_VEL
LIN {X 0,Y 387.106,Z 393.994,A -85,B 0,C 180,E1 -12133.657,E2 -12133.657} C_VEL
LIN {X 0,Y 386.289,Z 404.412,A -85,B 0,C 180,E1 -12134.637,E2 -12134.637} C_VEL
LIN {X 0,Y 385.531,Z 413.99,A -85,B 0,C 180,E1 -12135.754,E2 -12135.754} C_VEL
LIN {X 0,Y 384.623,Z 423.166,A -85,B 0,C 180,E1 -12137.066,E2 -12137.066} C_VEL
LIN {X 0,Y 383.725,Z 432.076,A -85,B 0,C 180,E1 -12138.646,E2 -12138.646} C_VEL
LIN {X 0,Y 383.019,Z 439.246,A -85,B 0,C 180,E1 -12140.229,E2 -12140.229} C_VEL
LIN {X 0,Y 382.522,Z 444.083,A -85,B 0,C 180,E1 -12141.549,E2 -12141.549} C_VEL
LIN {X 0,Y 382.11,Z 449.264,A -85,B 0,C 180,E1 -12143.317,E2 -12143.317} C_VEL
LIN {X 0,Y 381.96,Z 452.372,A -85,B 0,C 180,E1 -12144.722,E2 -12144.722} C_VEL
LIN {X 0,Y 381.756,Z 454.232,A -85,B 0,C 180,E1 -12145.778,E2 -12145.778} C_VEL
LIN {X 0,Y 381.682,Z 455.63,A -85,B 0,C 180,E1 -12146.834,E2 -12146.834} C_VEL
LIN {X 0,Y 381.667,Z 456.623,A -85,B 0,C 180,E1 -12147.89,E2 -12147.89} C_VEL
LIN {X 0,Y 381.64,Z 457.468,A -85,B 0,C 180,E1 -12150,E2 -12150} C_VEL
LIN {X 0,Y 381.644,Z 457.278,A -85,B 0,C 180,E1 -12151.056,E2 -12151.056} C_VEL
LIN {X 0,Y 381.667,Z 456.694,A -85,B 0,C 180,E1 -12152.111,E2 -12152.111} C_VEL
LIN {X 0,Y 381.753,Z 454.374,A -85,B 0,C 180,E1 -12154.223,E2 -12154.223} C_VEL
LIN {X 0,Y 382.023,Z 451.508,A -85,B 0,C 180,E1 -12155.808,E2 -12155.808} C_VEL
LIN {X 0,Y 382.26,Z 447.625,A -85,B 0,C 180,E1 -12157.395,E2 -12157.395} C_VEL
LIN {X 0,Y 382.694,Z 442.613,A -85,B 0,C 180,E1 -12158.981,E2 -12158.981} C_VEL
LIN {X 0,Y 383.321,Z 436.301,A -85,B 0,C 180,E1 -12160.565,E2 -12160.565} C_VEL
LIN {X 0,Y 384.07,Z 428.401,A -85,B 0,C 180,E1 -12162.148,E2 -12162.148} C_VEL
LIN {X 0,Y 385.099,Z 418.568,A -85,B 0,C 180,E1 -12163.724,E2 -12163.724} C_VEL
LIN {X 0,Y 386.021,Z 408.357,A -85,B 0,C 180,E1 -12165.024,E2 -12165.024} C_VEL
LIN {X 0,Y 386.754,Z 398.029,A -85,B 0,C 180,E1 -12166.088,E2 -12166.088} C_VEL
LIN {X 0,Y 387.791,Z 385.929,A -85,B 0,C 180,E1 -12167.062,E2 -12167.062} C_VEL
LIN {X 0,Y 388.006,Z 379.906,A -85,B 0,C 180,E1 -12167.463,E2 -12167.463} C_VEL
LIN {X 0,Y 385.625,Z 367.777,A -85,B 0,C 180,E1 -12168.241,E2 -12168.241} C_VEL
LIN {X 0,Y 382.391,Z 354.872,A -85,B 0,C 180,E1 -12168.89,E2 -12168.89} C_VEL
LIN {X 0,Y 382.265,Z 354.434,A -85,B 0,C 180,E1 -12168.91,E2 -12168.91} C_VEL
LIN {X 0,Y 381.663,Z 353.269,A -85,B 0,C 180,E1 -12169.069,E2 -12169.069} C_VEL
LIN {X 0,Y 378.802,Z 351.851,A -85,B 0,C 180,E1 -12170.19,E2 -12170.19} C_VEL
LIN {X 0,Y 376.309,Z 350.451,A -85,B 0,C 180,E1 -12171.759,E2 -12171.759} C_VEL
LIN {X 0,Y 375.413,Z 348.98,A -85,B 0,C 180,E1 -12172.778,E2 -12172.778} C_VEL
LIN {X 0,Y 375.22,Z 348.01,A -85,B 0,C 180,E1 -12173.464,E2 -12173.464} C_VEL
LIN {X 0,Y 375.41,Z 343.986,A -85,B 0,C 180,E1 -12176.699,E2 -12176.699} C_VEL
LIN {X 0,Y 375.677,Z 339.623,A -85,B 0,C 180,E1 -12180.338,E2 -12180.338} C_VEL
LIN {X 0,Y 375.85,Z 336.748,A -85,B 0,C 180,E1 -12182.838,E2 -12182.838} C_VEL
LIN {X 0,Y 375.898,Z 333.822,A -85,B 0,C 180,E1 -12185.422,E2 -12185.422} C_VEL
LIN {X 0,Y 375.88,Z 332.669,A -85,B 0,C 180,E1 -12186.487,E2 -12186.487} C_VEL
LIN {X 0,Y 375.96,Z 332.656,A -85,B 0,C 180,E1 -12189.463,E2 -12189.463} C_VEL
LIN {X 0,Y 375.934,Z 332.656,A -85,B 0,C 180,E1 -12193.189,E2 -12193.189} C_VEL
LIN {X 0,Y 375.931,Z 332.655,A -85,B 0,C 180,E1 -12196.811,E2 -12196.811} C_VEL
LIN {X 0,Y 375.933,Z 332.654,A -85,B 0,C 180,E1 -12200.533,E2 -12200.533} C_VEL
LIN {X 0,Y 375.961,Z 332.655,A -85,B 0,C 180,E1 -12203.495,E2 -12203.495} C_VEL
LIN {X 0,Y 375.958,Z 332.652,A -85,B 0,C 180,E1 -12205.888,E2 -12205.888} C_VEL
LIN {X 0,Y 375.959,Z 332.652,A -85,B 0,C 180,E1 -12209.687,E2 -12209.687} C_VEL
LIN {X 0,Y 375.925,Z 332.655,A -85,B 0,C 180,E1 -12212.135,E2 -12212.135} C_VEL
LIN {X 0,Y 375.969,Z 332.65,A -85,B 0,C 180,E1 -12215.717,E2 -12215.717} C_VEL
LIN {X 0,Y 375.995,Z 332.65,A -85,B 0,C 180,E1 -12219.198,E2 -12219.198} C_VEL
LIN {X 0,Y 376.047,Z 332.644,A -85,B 0,C 180,E1 -12222.601,E2 -12222.601} C_VEL
LIN {X 0,Y 376.086,Z 332.637,A -85,B 0,C 180,E1 -12226.342,E2 -12226.342} C_VEL
LIN {X 0,Y 376.115,Z 332.635,A -85,B 0,C 180,E1 -12230.318,E2 -12230.318} C_VEL
LIN {X 0,Y 376.227,Z 332.623,A -85,B 0,C 180,E1 -12232.486,E2 -12232.486} C_VEL
LIN {X 0,Y 376.168,Z 332.63,A -85,B 0,C 180,E1 -12234.64,E2 -12234.64} C_VEL
LIN {X 0,Y 376.347,Z 332.604,A -85,B 0,C 180,E1 -12237.86,E2 -12237.86} C_VEL
LIN {X 0,Y 376.453,Z 332.592,A -85,B 0,C 180,E1 -12240,E2 -12240} C_VEL
LIN {X 0,Y 376.346,Z 332.607,A -85,B 0,C 180,E1 -12242.14,E2 -12242.14} C_VEL
LIN {X 0,Y 376.238,Z 332.62,A -85,B 0,C 180,E1 -12246.435,E2 -12246.435} C_VEL
LIN {X 0,Y 376.115,Z 332.634,A -85,B 0,C 180,E1 -12249.682,E2 -12249.682} C_VEL
LIN {X 0,Y 376.086,Z 332.638,A -85,B 0,C 180,E1 -12253.658,E2 -12253.658} C_VEL
LIN {X 0,Y 376.04,Z 332.644,A -85,B 0,C 180,E1 -12257.607,E2 -12257.607} C_VEL
LIN {X 0,Y 375.975,Z 332.649,A -85,B 0,C 180,E1 -12260.832,E2 -12260.832} C_VEL
LIN {X 0,Y 375.972,Z 332.65,A -85,B 0,C 180,E1 -12264.283,E2 -12264.283} C_VEL
LIN {X 0,Y 375.926,Z 332.658,A -85,B 0,C 180,E1 -12267.864,E2 -12267.864} C_VEL
LIN {X 0,Y 375.955,Z 332.657,A -85,B 0,C 180,E1 -12271.562,E2 -12271.562} C_VEL
LIN {X 0,Y 375.956,Z 332.657,A -85,B 0,C 180,E1 -12275.416,E2 -12275.416} C_VEL
LIN {X 0,Y 375.935,Z 332.654,A -85,B 0,C 180,E1 -12278.264,E2 -12278.264} C_VEL
LIN {X 0,Y 375.911,Z 332.659,A -85,B 0,C 180,E1 -12281.597,E2 -12281.597} C_VEL
LIN {X 0,Y 375.921,Z 332.661,A -85,B 0,C 180,E1 -12284.731,E2 -12284.731} C_VEL
LIN {X 0,Y 375.981,Z 332.708,A -85,B 0,C 180,E1 -12287.264,E2 -12287.264} C_VEL
LIN {X 0,Y 376.845,Z 337.768,A -85,B 0,C 180,E1 -12290.648,E2 -12290.648} C_VEL
LIN {X 0,Y 377.392,Z 342.172,A -85,B 0,C 180,E1 -12293.422,E2 -12293.422} C_VEL
LIN {X 0,Y 377.283,Z 346.581,A -85,B 0,C 180,E1 -12296.025,E2 -12296.025} C_VEL
LIN {X 0,Y 376.873,Z 351.974,A -85,B 0,C 180,E1 -12299.073,E2 -12299.073} C_VEL
LIN {X 0,Y 376.275,Z 358.737,A -85,B 0,C 180,E1 -12302.767,E2 -12302.767} C_VEL
LIN {X 0,Y 375.776,Z 365.525,A -85,B 0,C 180,E1 -12306.41,E2 -12306.41} C_VEL
LIN {X 0,Y 375.479,Z 371.111,A -85,B 0,C 180,E1 -12309.37,E2 -12309.37} C_VEL
LIN {X 0,Y 375.328,Z 373.766,A -85,B 0,C 180,E1 -12310.712,E2 -12310.712} C_VEL
LIN {X 0,Y 377.876,Z 386.821,A -85,B 0,C 180,E1 -12311.284,E2 -12311.284} C_VEL
LIN {X 0,Y 379.661,Z 398.296,A -85,B 0,C 180,E1 -12311.954,E2 -12311.954} C_VEL
LIN {X 0,Y 380.612,Z 406.173,A -85,B 0,C 180,E1 -12312.511,E2 -12312.511} C_VEL
LIN {X 0,Y 379.639,Z 418.427,A -85,B 0,C 180,E1 -12313.463,E2 -12313.463} C_VEL
LIN {X 0,Y 378.599,Z 430.231,A -85,B 0,C 180,E1 -12314.661,E2 -12314.661} C_VEL
LIN {X 0,Y 377.598,Z 440.716,A -85,B 0,C 180,E1 -12315.997,E2 -12315.997} C_VEL
LIN {X 0,Y 376.777,Z 449.204,A -85,B 0,C 180,E1 -12317.339,E2 -12317.339} C_VEL
LIN {X 0,Y 375.957,Z 457.488,A -85,B 0,C 180,E1 -12318.953,E2 -12318.953} C_VEL
LIN {X 0,Y 375.35,Z 464.167,A -85,B 0,C 180,E1 -12320.57,E2 -12320.57} C_VEL
LIN {X 0,Y 374.891,Z 470.282,A -85,B 0,C 180,E1 -12322.459,E2 -12322.459} C_VEL
LIN {X 0,Y 374.671,Z 473.654,A -85,B 0,C 180,E1 -12323.808,E2 -12323.808} C_VEL
LIN {X 0,Y 374.569,Z 477.194,A -85,B 0,C 180,E1 -12325.695,E2 -12325.695} C_VEL
LIN {X 0,Y 374.458,Z 479.589,A -85,B 0,C 180,E1 -12327.848,E2 -12327.848} C_VEL
LIN {X 0,Y 374.491,Z 480.2,A -85,B 0,C 180,E1 -12328.924,E2 -12328.924} C_VEL
LIN {X 0,Y 374.508,Z 480.417,A -85,B 0,C 180,E1 -12330,E2 -12330} C_VEL
LIN {X 0,Y 374.491,Z 480.2,A -85,B 0,C 180,E1 -12331.075,E2 -12331.075} C_VEL
LIN {X 0,Y 374.462,Z 478.592,A -85,B 0,C 180,E1 -12333.227,E2 -12333.227} C_VEL
LIN {X 0,Y 374.568,Z 477.195,A -85,B 0,C 180,E1 -12334.304,E2 -12334.304} C_VEL
LIN {X 0,Y 374.664,Z 473.671,A -85,B 0,C 180,E1 -12336.182,E2 -12336.182} C_VEL
LIN {X 0,Y 374.981,Z 468.68,A -85,B 0,C 180,E1 -12338.08,E2 -12338.08} C_VEL
LIN {X 0,Y 375.459,Z 463.147,A -85,B 0,C 180,E1 -12339.698,E2 -12339.698} C_VEL
LIN {X 0,Y 376.05,Z 456.24,A -85,B 0,C 180,E1 -12341.316,E2 -12341.316} C_VEL
LIN {X 0,Y 376.982,Z 447.606,A -85,B 0,C 180,E1 -12342.927,E2 -12342.927} C_VEL
LIN {X 0,Y 377.937,Z 437.697,A -85,B 0,C 180,E1 -12344.411,E2 -12344.411} C_VEL
LIN {X 0,Y 378.78,Z 427.852,A -85,B 0,C 180,E1 -12345.606,E2 -12345.606} C_VEL
LIN {X 0,Y 379.795,Z 416.862,A -85,B 0,C 180,E1 -12346.667,E2 -12346.667} C_VEL
LIN {X 0,Y 380.576,Z 406.132,A -85,B 0,C 180,E1 -12347.49,E2 -12347.49} C_VEL
LIN {X 0,Y 379.031,Z 393.993,A -85,B 0,C 180,E1 -12348.309,E2 -12348.309} C_VEL
LIN {X 0,Y 376.873,Z 381.406,A -85,B 0,C 180,E1 -12348.973,E2 -12348.973} C_VEL
LIN {X 0,Y 375.327,Z 373.602,A -85,B 0,C 180,E1 -12349.305,E2 -12349.305} C_VEL
LIN {X 0,Y 375.735,Z 366.391,A -85,B 0,C 180,E1 -12353.128,E2 -12353.128} C_VEL
LIN {X 0,Y 376.198,Z 359.826,A -85,B 0,C 180,E1 -12356.637,E2 -12356.637} C_VEL
LIN {X 0,Y 376.72,Z 353.189,A -85,B 0,C 180,E1 -12360.244,E2 -12360.244} C_VEL
LIN {X 0,Y 377.175,Z 348.214,A -85,B 0,C 180,E1 -12363.018,E2 -12363.018} C_VEL
LIN {X 0,Y 377.436,Z 343.238,A -85,B 0,C 180,E1 -12365.911,E2 -12365.911} C_VEL
LIN {X 0,Y 377.096,Z 339.079,A -85,B 0,C 180,E1 -12368.486,E2 -12368.486} C_VEL
LIN {X 0,Y 376.321,Z 334.236,A -85,B 0,C 180,E1 -12371.667,E2 -12371.667} C_VEL
LIN {X 0,Y 376.025,Z 332.651,A -85,B 0,C 180,E1 -12372.864,E2 -12372.864} C_VEL
LIN {X 0,Y 375.93,Z 332.658,A -85,B 0,C 180,E1 -12376.234,E2 -12376.234} C_VEL
LIN {X 0,Y 375.934,Z 332.654,A -85,B 0,C 180,E1 -12380.037,E2 -12380.037} C_VEL
LIN {X 0,Y 375.957,Z 332.651,A -85,B 0,C 180,E1 -12383.495,E2 -12383.495} C_VEL
LIN {X 0,Y 375.953,Z 332.652,A -85,B 0,C 180,E1 -12385.888,E2 -12385.888} C_VEL
LIN {X 0,Y 375.953,Z 332.652,A -85,B 0,C 180,E1 -12389.686,E2 -12389.686} C_VEL
LIN {X 0,Y 375.921,Z 332.659,A -85,B 0,C 180,E1 -12392.135,E2 -12392.135} C_VEL
LIN {X 0,Y 375.966,Z 332.651,A -85,B 0,C 180,E1 -12395.717,E2 -12395.717} C_VEL
LIN {X 0,Y 375.989,Z 332.647,A -85,B 0,C 180,E1 -12399.197,E2 -12399.197} C_VEL
LIN {X 0,Y 376.041,Z 332.643,A -85,B 0,C 180,E1 -12402.601,E2 -12402.601} C_VEL
LIN {X 0,Y 376.08,Z 332.639,A -85,B 0,C 180,E1 -12406.342,E2 -12406.342} C_VEL
LIN {X 0,Y 376.109,Z 332.635,A -85,B 0,C 180,E1 -12410.318,E2 -12410.318} C_VEL
LIN {X 0,Y 376.221,Z 332.619,A -85,B 0,C 180,E1 -12412.486,E2 -12412.486} C_VEL
LIN {X 0,Y 376.169,Z 332.625,A -85,B 0,C 180,E1 -12414.64,E2 -12414.64} C_VEL
LIN {X 0,Y 376.344,Z 332.608,A -85,B 0,C 180,E1 -12417.86,E2 -12417.86} C_VEL
LIN {X 0,Y 376.449,Z 332.593,A -85,B 0,C 180,E1 -12420,E2 -12420} C_VEL
LIN {X 0,Y 376.341,Z 332.605,A -85,B 0,C 180,E1 -12422.141,E2 -12422.141} C_VEL
LIN {X 0,Y 376.229,Z 332.617,A -85,B 0,C 180,E1 -12426.574,E2 -12426.574} C_VEL
LIN {X 0,Y 376.196,Z 332.621,A -85,B 0,C 180,E1 -12428.595,E2 -12428.595} C_VEL
LIN {X 0,Y 376.04,Z 332.642,A -85,B 0,C 180,E1 -12431.864,E2 -12431.864} C_VEL
LIN {X 0,Y 376.048,Z 332.645,A -85,B 0,C 180,E1 -12435.168,E2 -12435.168} C_VEL
LIN {X 0,Y 376,Z 332.646,A -85,B 0,C 180,E1 -12438.527,E2 -12438.527} C_VEL
LIN {X 0,Y 375.95,Z 332.652,A -85,B 0,C 180,E1 -12441.955,E2 -12441.955} C_VEL
LIN {X 0,Y 375.967,Z 332.65,A -85,B 0,C 180,E1 -12444.283,E2 -12444.283} C_VEL
LIN {X 0,Y 375.92,Z 332.656,A -85,B 0,C 180,E1 -12447.865,E2 -12447.865} C_VEL
LIN {X 0,Y 375.949,Z 332.652,A -85,B 0,C 180,E1 -12451.563,E2 -12451.563} C_VEL
LIN {X 0,Y 375.951,Z 332.653,A -85,B 0,C 180,E1 -12455.416,E2 -12455.416} C_VEL
LIN {X 0,Y 375.93,Z 332.657,A -85,B 0,C 180,E1 -12458.264,E2 -12458.264} C_VEL
LIN {X 0,Y 375.911,Z 332.657,A -85,B 0,C 180,E1 -12461.599,E2 -12461.599} C_VEL
LIN {X 0,Y 375.921,Z 332.659,A -85,B 0,C 180,E1 -12464.732,E2 -12464.732} C_VEL
LIN {X 0,Y 375.957,Z 332.657,A -85,B 0,C 180,E1 -12468.396,E2 -12468.396} C_VEL
LIN {X 0,Y 375.968,Z 332.651,A -85,B 0,C 180,E1 -12471.731,E2 -12471.731} C_VEL
LIN {X 0,Y 375.873,Z 332.668,A -85,B 0,C 180,E1 -12473.515,E2 -12473.515} C_VEL
LIN {X 0,Y 375.902,Z 335.162,A -85,B 0,C 180,E1 -12475.884,E2 -12475.884} C_VEL
LIN {X 0,Y 375.69,Z 339.516,A -85,B 0,C 180,E1 -12479.664,E2 -12479.664} C_VEL
LIN {X 0,Y 375.412,Z 343.848,A -85,B 0,C 180,E1 -12483.302,E2 -12483.302} C_VEL
LIN {X 0,Y 375.234,Z 348.247,A -85,B 0,C 180,E1 -12486.84,E2 -12486.84} C_VEL
LIN {X 0,Y 375.031,Z 353.395,A -85,B 0,C 180,E1 -12490.776,E2 -12490.776} C_VEL
LIN {X 0,Y 378.359,Z 366.673,A -85,B 0,C 180,E1 -12491.435,E2 -12491.435} C_VEL
LIN {X 0,Y 380.787,Z 378.463,A -85,B 0,C 180,E1 -12492.193,E2 -12492.193} C_VEL
LIN {X 0,Y 381.186,Z 382.589,A -85,B 0,C 180,E1 -12492.483,E2 -12492.483} C_VEL
LIN {X 0,Y 380.302,Z 394.215,A -85,B 0,C 180,E1 -12493.356,E2 -12493.356} C_VEL
LIN {X 0,Y 379.398,Z 405.268,A -85,B 0,C 180,E1 -12494.42,E2 -12494.42} C_VEL
LIN {X 0,Y 378.666,Z 414.209,A -85,B 0,C 180,E1 -12495.49,E2 -12495.49} C_VEL
LIN {X 0,Y 377.687,Z 423.385,A -85,B 0,C 180,E1 -12496.824,E2 -12496.824} C_VEL
LIN {X 0,Y 376.769,Z 432.293,A -85,B 0,C 180,E1 -12498.433,E2 -12498.433} C_VEL
LIN {X 0,Y 376.027,Z 439.464,A -85,B 0,C 180,E1 -12500.045,E2 -12500.045} C_VEL
LIN {X 0,Y 375.506,Z 444.3,A -85,B 0,C 180,E1 -12501.389,E2 -12501.389} C_VEL
LIN {X 0,Y 375.046,Z 449.753,A -85,B 0,C 180,E1 -12503.302,E2 -12503.302} C_VEL
LIN {X 0,Y 374.885,Z 452.589,A -85,B 0,C 180,E1 -12504.622,E2 -12504.622} C_VEL
LIN {X 0,Y 374.689,Z 454.448,A -85,B 0,C 180,E1 -12505.698,E2 -12505.698} C_VEL
LIN {X 0,Y 374.591,Z 455.846,A -85,B 0,C 180,E1 -12506.774,E2 -12506.774} C_VEL
LIN {X 0,Y 374.561,Z 457.45,A -85,B 0,C 180,E1 -12508.925,E2 -12508.925} C_VEL
LIN {X 0,Y 374.555,Z 457.683,A -85,B 0,C 180,E1 -12510,E2 -12510} C_VEL
LIN {X 0,Y 374.562,Z 457.493,A -85,B 0,C 180,E1 -12511.076,E2 -12511.076} C_VEL
LIN {X 0,Y 374.589,Z 455.944,A -85,B 0,C 180,E1 -12513.227,E2 -12513.227} C_VEL
LIN {X 0,Y 374.686,Z 454.589,A -85,B 0,C 180,E1 -12514.303,E2 -12514.303} C_VEL
LIN {X 0,Y 374.964,Z 451.722,A -85,B 0,C 180,E1 -12515.917,E2 -12515.917} C_VEL
LIN {X 0,Y 375.198,Z 447.84,A -85,B 0,C 180,E1 -12517.535,E2 -12517.535} C_VEL
LIN {X 0,Y 375.673,Z 442.827,A -85,B 0,C 180,E1 -12519.15,E2 -12519.15} C_VEL
LIN {X 0,Y 376.334,Z 436.515,A -85,B 0,C 180,E1 -12520.763,E2 -12520.763} C_VEL
LIN {X 0,Y 377.132,Z 428.613,A -85,B 0,C 180,E1 -12522.375,E2 -12522.375} C_VEL
LIN {X 0,Y 378.209,Z 418.78,A -85,B 0,C 180,E1 -12523.979,E2 -12523.979} C_VEL
LIN {X 0,Y 379.164,Z 408.568,A -85,B 0,C 180,E1 -12525.303,E2 -12525.303} C_VEL
LIN {X 0,Y 379.95,Z 398.239,A -85,B 0,C 180,E1 -12526.385,E2 -12526.385} C_VEL
LIN {X 0,Y 380.996,Z 386.266,A -85,B 0,C 180,E1 -12527.366,E2 -12527.366} C_VEL
LIN {X 0,Y 381.126,Z 380.586,A -85,B 0,C 180,E1 -12527.759,E2 -12527.759} C_VEL
LIN {X 0,Y 378.664,Z 368.016,A -85,B 0,C 180,E1 -12528.588,E2 -12528.588} C_VEL
LIN {X 0,Y 375.367,Z 355.173,A -85,B 0,C 180,E1 -12529.254,E2 -12529.254} C_VEL
LIN {X 0,Y 375.007,Z 353.338,A -85,B 0,C 180,E1 -12529.358,E2 -12529.358} C_VEL
LIN {X 0,Y 375.199,Z 348.391,A -85,B 0,C 180,E1 -12533.164,E2 -12533.164} C_VEL
LIN {X 0,Y 375.22,Z 348.01,A -85,B 0,C 180,E1 -12533.464,E2 -12533.464} C_VEL
LIN {X 0,Y 374.562,Z 346.986,A -85,B 0,C 180,E1 -12534.347,E2 -12534.347} C_VEL
LIN {X 0,Y 371.768,Z 345.527,A -85,B 0,C 180,E1 -12535.792,E2 -12535.792} C_VEL
LIN {X 0,Y 369.448,Z 344.392,A -85,B 0,C 180,E1 -12536.96,E2 -12536.96} C_VEL
LIN {X 0,Y 368.512,Z 343.427,A -85,B 0,C 180,E1 -12537.86,E2 -12537.86} C_VEL
LIN {X 0,Y 368.467,Z 343.072,A -85,B 0,C 180,E1 -12538.163,E2 -12538.163} C_VEL
LIN {X 0,Y 368.685,Z 339.808,A -85,B 0,C 180,E1 -12540.976,E2 -12540.976} C_VEL
LIN {X 0,Y 368.833,Z 336.881,A -85,B 0,C 180,E1 -12543.544,E2 -12543.544} C_VEL
LIN {X 0,Y 368.846,Z 333.961,A -85,B 0,C 180,E1 -12546.205,E2 -12546.205} C_VEL
LIN {X 0,Y 368.842,Z 333.546,A -85,B 0,C 180,E1 -12546.843,E2 -12546.843} C_VEL
LIN {X 0,Y 368.899,Z 333.535,A -85,B 0,C 180,E1 -12548.953,E2 -12548.953} C_VEL
LIN {X 0,Y 368.881,Z 333.535,A -85,B 0,C 180,E1 -12552.009,E2 -12552.009} C_VEL
LIN {X 0,Y 368.875,Z 333.535,A -85,B 0,C 180,E1 -12555.175,E2 -12555.175} C_VEL
LIN {X 0,Y 368.858,Z 333.536,A -85,B 0,C 180,E1 -12558.174,E2 -12558.174} C_VEL
LIN {X 0,Y 368.875,Z 333.539,A -85,B 0,C 180,E1 -12561.366,E2 -12561.366} C_VEL
LIN {X 0,Y 368.935,Z 333.53,A -85,B 0,C 180,E1 -12565.146,E2 -12565.146} C_VEL
LIN {X 0,Y 368.91,Z 333.533,A -85,B 0,C 180,E1 -12569.045,E2 -12569.045} C_VEL
LIN {X 0,Y 368.909,Z 333.531,A -85,B 0,C 180,E1 -12571.558,E2 -12571.558} C_VEL
LIN {X 0,Y 368.922,Z 333.531,A -85,B 0,C 180,E1 -12575.222,E2 -12575.222} C_VEL
LIN {X 0,Y 368.917,Z 333.534,A -85,B 0,C 180,E1 -12578.98,E2 -12578.98} C_VEL
LIN {X 0,Y 368.988,Z 333.52,A -85,B 0,C 180,E1 -12582.257,E2 -12582.257} C_VEL
LIN {X 0,Y 369.034,Z 333.515,A -85,B 0,C 180,E1 -12586.228,E2 -12586.228} C_VEL
LIN {X 0,Y 369.064,Z 333.511,A -85,B 0,C 180,E1 -12590.132,E2 -12590.132} C_VEL
LIN {X 0,Y 369.185,Z 333.498,A -85,B 0,C 180,E1 -12592.342,E2 -12592.342} C_VEL
LIN {X 0,Y 369.141,Z 333.506,A -85,B 0,C 180,E1 -12594.537,E2 -12594.537} C_VEL
LIN {X 0,Y 369.312,Z 333.48,A -85,B 0,C 180,E1 -12597.819,E2 -12597.819} C_VEL
LIN {X 0,Y 369.404,Z 333.47,A -85,B 0,C 180,E1 -12600,E2 -12600} C_VEL
LIN {X 0,Y 369.312,Z 333.484,A -85,B 0,C 180,E1 -12602.181,E2 -12602.181} C_VEL
LIN {X 0,Y 369.198,Z 333.495,A -85,B 0,C 180,E1 -12606.558,E2 -12606.558} C_VEL
LIN {X 0,Y 369.064,Z 333.514,A -85,B 0,C 180,E1 -12609.868,E2 -12609.868} C_VEL
LIN {X 0,Y 369.034,Z 333.517,A -85,B 0,C 180,E1 -12613.772,E2 -12613.772} C_VEL
LIN {X 0,Y 368.998,Z 333.523,A -85,B 0,C 180,E1 -12617.769,E2 -12617.769} C_VEL
LIN {X 0,Y 368.907,Z 333.53,A -85,B 0,C 180,E1 -12621.221,E2 -12621.221} C_VEL
LIN {X 0,Y 368.925,Z 333.527,A -85,B 0,C 180,E1 -12624.778,E2 -12624.778} C_VEL
LIN {X 0,Y 368.894,Z 333.531,A -85,B 0,C 180,E1 -12628.793,E2 -12628.793} C_VEL
LIN {X 0,Y 368.896,Z 333.531,A -85,B 0,C 180,E1 -12632.238,E2 -12632.238} C_VEL
LIN {X 0,Y 368.927,Z 333.529,A -85,B 0,C 180,E1 -12635.002,E2 -12635.002} C_VEL
LIN {X 0,Y 368.876,Z 333.534,A -85,B 0,C 180,E1 -12638.635,E2 -12638.635} C_VEL
LIN {X 0,Y 368.856,Z 333.536,A -85,B 0,C 180,E1 -12642.005,E2 -12642.005} C_VEL
LIN {X 0,Y 368.876,Z 333.539,A -85,B 0,C 180,E1 -12645.176,E2 -12645.176} C_VEL
LIN {X 0,Y 368.923,Z 333.612,A -85,B 0,C 180,E1 -12646.944,E2 -12646.944} C_VEL
LIN {X 0,Y 369.821,Z 338.738,A -85,B 0,C 180,E1 -12650.46,E2 -12650.46} C_VEL
LIN {X 0,Y 370.32,Z 342.436,A -85,B 0,C 180,E1 -12652.853,E2 -12652.853} C_VEL
LIN {X 0,Y 370.36,Z 346.435,A -85,B 0,C 180,E1 -12655.3,E2 -12655.3} C_VEL
LIN {X 0,Y 369.999,Z 350.839,A -85,B 0,C 180,E1 -12657.87,E2 -12657.87} C_VEL
LIN {X 0,Y 369.451,Z 356.483,A -85,B 0,C 180,E1 -12661.051,E2 -12661.051} C_VEL
LIN {X 0,Y 368.944,Z 362.928,A -85,B 0,C 180,E1 -12664.621,E2 -12664.621} C_VEL
LIN {X 0,Y 368.516,Z 369.451,A -85,B 0,C 180,E1 -12668.168,E2 -12668.168} C_VEL
LIN {X 0,Y 368.283,Z 373.557,A -85,B 0,C 180,E1 -12670.328,E2 -12670.328} C_VEL
LIN {X 0,Y 370.944,Z 386.859,A -85,B 0,C 180,E1 -12670.933,E2 -12670.933} C_VEL
LIN {X 0,Y 372.843,Z 399.422,A -85,B 0,C 180,E1 -12671.697,E2 -12671.697} C_VEL
LIN {X 0,Y 373.736,Z 407.555,A -85,B 0,C 180,E1 -12672.292,E2 -12672.292} C_VEL
LIN {X 0,Y 372.712,Z 419.645,A -85,B 0,C 180,E1 -12673.288,E2 -12673.288} C_VEL
LIN {X 0,Y 371.619,Z 431.196,A -85,B 0,C 180,E1 -12674.506,E2 -12674.506} C_VEL
LIN {X 0,Y 370.693,Z 440.503,A -85,B 0,C 180,E1 -12675.731,E2 -12675.731} C_VEL
LIN {X 0,Y 369.831,Z 448.99,A -85,B 0,C 180,E1 -12677.098,E2 -12677.098} C_VEL
LIN {X 0,Y 368.932,Z 457.272,A -85,B 0,C 180,E1 -12678.74,E2 -12678.74} C_VEL
LIN {X 0,Y 368.311,Z 463.951,A -85,B 0,C 180,E1 -12680.388,E2 -12680.388} C_VEL
LIN {X 0,Y 367.812,Z 470.066,A -85,B 0,C 180,E1 -12682.313,E2 -12682.313} C_VEL
LIN {X 0,Y 367.563,Z 473.835,A -85,B 0,C 180,E1 -12683.864,E2 -12683.864} C_VEL
LIN {X 0,Y 367.475,Z 476.979,A -85,B 0,C 180,E1 -12685.612,E2 -12685.612} C_VEL
LIN {X 0,Y 367.358,Z 479.374,A -85,B 0,C 180,E1 -12687.807,E2 -12687.807} C_VEL
LIN {X 0,Y 367.392,Z 479.984,A -85,B 0,C 180,E1 -12688.903,E2 -12688.903} C_VEL
LIN {X 0,Y 367.411,Z 480.202,A -85,B 0,C 180,E1 -12690,E2 -12690} C_VEL
LIN {X 0,Y 367.392,Z 479.984,A -85,B 0,C 180,E1 -12691.096,E2 -12691.096} C_VEL
LIN {X 0,Y 367.381,Z 478.376,A -85,B 0,C 180,E1 -12693.289,E2 -12693.289} C_VEL
LIN {X 0,Y 367.475,Z 476.979,A -85,B 0,C 180,E1 -12694.387,E2 -12694.387} C_VEL
LIN {X 0,Y 367.557,Z 473.849,A -85,B 0,C 180,E1 -12696.127,E2 -12696.127} C_VEL
LIN {X 0,Y 367.798,Z 470.057,A -85,B 0,C 180,E1 -12697.686,E2 -12697.686} C_VEL
LIN {X 0,Y 368.317,Z 463.942,A -85,B 0,C 180,E1 -12699.611,E2 -12699.611} C_VEL
LIN {X 0,Y 368.932,Z 457.26,A -85,B 0,C 180,E1 -12701.259,E2 -12701.259} C_VEL
LIN {X 0,Y 369.842,Z 448.974,A -85,B 0,C 180,E1 -12702.901,E2 -12702.901} C_VEL
LIN {X 0,Y 370.719,Z 440.482,A -85,B 0,C 180,E1 -12704.267,E2 -12704.267} C_VEL
LIN {X 0,Y 371.706,Z 429.989,A -85,B 0,C 180,E1 -12705.63,E2 -12705.63} C_VEL
LIN {X 0,Y 372.683,Z 419.611,A -85,B 0,C 180,E1 -12706.712,E2 -12706.712} C_VEL
LIN {X 0,Y 373.733,Z 407.513,A -85,B 0,C 180,E1 -12707.706,E2 -12707.706} C_VEL
LIN {X 0,Y 372.331,Z 395.744,A -85,B 0,C 180,E1 -12708.543,E2 -12708.543} C_VEL
LIN {X 0,Y 370.201,Z 383.005,A -85,B 0,C 180,E1 -12709.257,E2 -12709.257} C_VEL
LIN {X 0,Y 368.286,Z 373.394,A -85,B 0,C 180,E1 -12709.689,E2 -12709.689} C_VEL
LIN {X 0,Y 368.661,Z 367.288,A -85,B 0,C 180,E1 -12713.003,E2 -12713.003} C_VEL
LIN {X 0,Y 369.111,Z 360.873,A -85,B 0,C 180,E1 -12716.505,E2 -12716.505} C_VEL
LIN {X 0,Y 369.679,Z 354.132,A -85,B 0,C 180,E1 -12720.25,E2 -12720.25} C_VEL
LIN {X 0,Y 370.176,Z 348.604,A -85,B 0,C 180,E1 -12723.406,E2 -12723.406} C_VEL
LIN {X 0,Y 370.432,Z 344.192,A -85,B 0,C 180,E1 -12726.024,E2 -12726.024} C_VEL
LIN {X 0,Y 370.001,Z 339.741,A -85,B 0,C 180,E1 -12728.851,E2 -12728.851} C_VEL
LIN {X 0,Y 369.278,Z 334.962,A -85,B 0,C 180,E1 -12732.077,E2 -12732.077} C_VEL
LIN {X 0,Y 368.972,Z 333.532,A -85,B 0,C 180,E1 -12733.125,E2 -12733.125} C_VEL
LIN {X 0,Y 368.883,Z 333.537,A -85,B 0,C 180,E1 -12736.695,E2 -12736.695} C_VEL
LIN {X 0,Y 368.878,Z 333.533,A -85,B 0,C 180,E1 -12739.647,E2 -12739.647} C_VEL
LIN {X 0,Y 368.894,Z 333.532,A -85,B 0,C 180,E1 -12743.143,E2 -12743.143} C_VEL
LIN {X 0,Y 368.889,Z 333.536,A -85,B 0,C 180,E1 -12746.461,E2 -12746.461} C_VEL
LIN {X 0,Y 368.905,Z 333.531,A -85,B 0,C 180,E1 -12749.044,E2 -12749.044} C_VEL
LIN {X 0,Y 368.904,Z 333.529,A -85,B 0,C 180,E1 -12751.557,E2 -12751.557} C_VEL
LIN {X 0,Y 368.919,Z 333.528,A -85,B 0,C 180,E1 -12755.222,E2 -12755.222} C_VEL
LIN {X 0,Y 368.901,Z 333.531,A -85,B 0,C 180,E1 -12758.779,E2 -12758.779} C_VEL
LIN {X 0,Y 368.982,Z 333.525,A -85,B 0,C 180,E1 -12762.257,E2 -12762.257} C_VEL
LIN {X 0,Y 369.028,Z 333.518,A -85,B 0,C 180,E1 -12766.228,E2 -12766.228} C_VEL
LIN {X 0,Y 369.058,Z 333.515,A -85,B 0,C 180,E1 -12770.131,E2 -12770.131} C_VEL
LIN {X 0,Y 369.179,Z 333.497,A -85,B 0,C 180,E1 -12772.342,E2 -12772.342} C_VEL
LIN {X 0,Y 369.142,Z 333.5,A -85,B 0,C 180,E1 -12774.538,E2 -12774.538} C_VEL
LIN {X 0,Y 369.309,Z 333.485,A -85,B 0,C 180,E1 -12777.819,E2 -12777.819} C_VEL
LIN {X 0,Y 369.399,Z 333.471,A -85,B 0,C 180,E1 -12780,E2 -12780} C_VEL
LIN {X 0,Y 369.307,Z 333.48,A -85,B 0,C 180,E1 -12782.181,E2 -12782.181} C_VEL
LIN {X 0,Y 369.2,Z 333.492,A -85,B 0,C 180,E1 -12786.561,E2 -12786.561} C_VEL
LIN {X 0,Y 369.128,Z 333.502,A -85,B 0,C 180,E1 -12788.761,E2 -12788.761} C_VEL
LIN {X 0,Y 368.995,Z 333.518,A -85,B 0,C 180,E1 -12792.094,E2 -12792.094} C_VEL
LIN {X 0,Y 368.988,Z 333.523,A -85,B 0,C 180,E1 -12795.465,E2 -12795.465} C_VEL
LIN {X 0,Y 368.949,Z 333.527,A -85,B 0,C 180,E1 -12798.895,E2 -12798.895} C_VEL
LIN {X 0,Y 368.917,Z 333.528,A -85,B 0,C 180,E1 -12802.396,E2 -12802.396} C_VEL
LIN {X 0,Y 368.918,Z 333.528,A -85,B 0,C 180,E1 -12805.986,E2 -12805.986} C_VEL
LIN {X 0,Y 368.887,Z 333.532,A -85,B 0,C 180,E1 -12809.693,E2 -12809.693} C_VEL
LIN {X 0,Y 368.89,Z 333.535,A -85,B 0,C 180,E1 -12813.044,E2 -12813.044} C_VEL
LIN {X 0,Y 368.91,Z 333.53,A -85,B 0,C 180,E1 -12816.198,E2 -12816.198} C_VEL
LIN {X 0,Y 368.868,Z 333.537,A -85,B 0,C 180,E1 -12818.958,E2 -12818.958} C_VEL
LIN {X 0,Y 368.864,Z 333.535,A -85,B 0,C 180,E1 -12822.008,E2 -12822.008} C_VEL
LIN {X 0,Y 368.874,Z 333.534,A -85,B 0,C 180,E1 -12825.177,E2 -12825.177} C_VEL
LIN {X 0,Y 368.906,Z 333.533,A -85,B 0,C 180,E1 -12828.182,E2 -12828.182} C_VEL
LIN {X 0,Y 368.905,Z 333.529,A -85,B 0,C 180,E1 -12831.361,E2 -12831.361} C_VEL
LIN {X 0,Y 368.837,Z 333.544,A -85,B 0,C 180,E1 -12833.158,E2 -12833.158} C_VEL
LIN {X 0,Y 368.84,Z 333.854,A -85,B 0,C 180,E1 -12833.796,E2 -12833.796} C_VEL
LIN {X 0,Y 368.826,Z 336.787,A -85,B 0,C 180,E1 -12836.456,E2 -12836.456} C_VEL
LIN {X 0,Y 368.684,Z 339.723,A -85,B 0,C 180,E1 -12839.072,E2 -12839.072} C_VEL
LIN {X 0,Y 368.514,Z 342.574,A -85,B 0,C 180,E1 -12841.526,E2 -12841.526} C_VEL
LIN {X 0,Y 368.368,Z 345.495,A -85,B 0,C 180,E1 -12843.973,E2 -12843.973} C_VEL
LIN {X 0,Y 368.096,Z 349.927,A -85,B 0,C 180,E1 -12847.552,E2 -12847.552} C_VEL
LIN {X 0,Y 368.004,Z 353.673,A -85,B 0,C 180,E1 -12850.395,E2 -12850.395} C_VEL
LIN {X 0,Y 371.332,Z 366.835,A -85,B 0,C 180,E1 -12851.067,E2 -12851.067} C_VEL
LIN {X 0,Y 373.92,Z 379.23,A -85,B 0,C 180,E1 -12851.888,E2 -12851.888} C_VEL
LIN {X 0,Y 374.42,Z 383.082,A -85,B 0,C 180,E1 -12852.175,E2 -12852.175} C_VEL
LIN {X 0,Y 373.515,Z 394.436,A -85,B 0,C 180,E1 -12853.044,E2 -12853.044} C_VEL
LIN {X 0,Y 372.632,Z 404.513,A -85,B 0,C 180,E1 -12854.022,E2 -12854.022} C_VEL
LIN {X 0,Y 371.814,Z 414.428,A -85,B 0,C 180,E1 -12855.217,E2 -12855.217} C_VEL
LIN {X 0,Y 370.773,Z 423.604,A -85,B 0,C 180,E1 -12856.574,E2 -12856.574} C_VEL
LIN {X 0,Y 369.818,Z 432.511,A -85,B 0,C 180,E1 -12858.213,E2 -12858.213} C_VEL
LIN {X 0,Y 369.046,Z 439.681,A -85,B 0,C 180,E1 -12859.855,E2 -12859.855} C_VEL
LIN {X 0,Y 368.479,Z 444.517,A -85,B 0,C 180,E1 -12861.224,E2 -12861.224} C_VEL
LIN {X 0,Y 368.045,Z 449.215,A -85,B 0,C 180,E1 -12862.871,E2 -12862.871} C_VEL
LIN {X 0,Y 367.817,Z 452.805,A -85,B 0,C 180,E1 -12864.518,E2 -12864.518} C_VEL
LIN {X 0,Y 367.624,Z 454.664,A -85,B 0,C 180,E1 -12865.615,E2 -12865.615} C_VEL
LIN {X 0,Y 367.504,Z 456.062,A -85,B 0,C 180,E1 -12866.712,E2 -12866.712} C_VEL
LIN {X 0,Y 367.465,Z 457.666,A -85,B 0,C 180,E1 -12868.905,E2 -12868.905} C_VEL
LIN {X 0,Y 367.458,Z 457.898,A -85,B 0,C 180,E1 -12870,E2 -12870} C_VEL
LIN {X 0,Y 367.465,Z 457.708,A -85,B 0,C 180,E1 -12871.096,E2 -12871.096} C_VEL
LIN {X 0,Y 367.503,Z 456.159,A -85,B 0,C 180,E1 -12873.289,E2 -12873.289} C_VEL
LIN {X 0,Y 367.622,Z 454.803,A -85,B 0,C 180,E1 -12874.386,E2 -12874.386} C_VEL
LIN {X 0,Y 367.907,Z 451.936,A -85,B 0,C 180,E1 -12876.031,E2 -12876.031} C_VEL
LIN {X 0,Y 368.159,Z 448.054,A -85,B 0,C 180,E1 -12877.68,E2 -12877.68} C_VEL
LIN {X 0,Y 368.669,Z 443.041,A -85,B 0,C 180,E1 -12879.325,E2 -12879.325} C_VEL
LIN {X 0,Y 369.351,Z 436.728,A -85,B 0,C 180,E1 -12880.969,E2 -12880.969} C_VEL
LIN {X 0,Y 370.181,Z 428.826,A -85,B 0,C 180,E1 -12882.611,E2 -12882.611} C_VEL
LIN {X 0,Y 371.321,Z 418.992,A -85,B 0,C 180,E1 -12884.244,E2 -12884.244} C_VEL
LIN {X 0,Y 372.304,Z 408.888,A -85,B 0,C 180,E1 -12885.579,E2 -12885.579} C_VEL
LIN {X 0,Y 373.144,Z 398.449,A -85,B 0,C 180,E1 -12886.692,E2 -12886.692} C_VEL
LIN {X 0,Y 374.225,Z 386.587,A -85,B 0,C 180,E1 -12887.681,E2 -12887.681} C_VEL
LIN {X 0,Y 374.259,Z 381.195,A -85,B 0,C 180,E1 -12888.069,E2 -12888.069} C_VEL
LIN {X 0,Y 371.74,Z 368.666,A -85,B 0,C 180,E1 -12888.926,E2 -12888.926} C_VEL
LIN {X 0,Y 368.386,Z 355.556,A -85,B 0,C 180,E1 -12889.628,E2 -12889.628} C_VEL
LIN {X 0,Y 367.98,Z 353.54,A -85,B 0,C 180,E1 -12889.746,E2 -12889.746} C_VEL
LIN {X 0,Y 368.173,Z 348.589,A -85,B 0,C 180,E1 -12893.632,E2 -12893.632} C_VEL
LIN {X 0,Y 368.401,Z 344.172,A -85,B 0,C 180,E1 -12897.248,E2 -12897.248} C_VEL
LIN {X 0,Y 368.467,Z 343.072,A -85,B 0,C 180,E1 -12898.163,E2 -12898.163} C_VEL
LIN {X 0,Y 367.906,Z 342.091,A -85,B 0,C 180,E1 -12899.064,E2 -12899.064} C_VEL
LIN {X 0,Y 365.176,Z 340.761,A -85,B 0,C 180,E1 -12900.539,E2 -12900.539} C_VEL
LIN {X 0,Y 362.829,Z 339.708,A -85,B 0,C 180,E1 -12901.733,E2 -12901.733} C_VEL
LIN {X 0,Y 361.839,Z 338.808,A -85,B 0,C 180,E1 -12902.652,E2 -12902.652} C_VEL
LIN {X 0,Y 361.771,Z 338.475,A -85,B 0,C 180,E1 -12902.962,E2 -12902.962} C_VEL
LIN {X 0,Y 361.821,Z 335.589,A -85,B 0,C 180,E1 -12905.642,E2 -12905.642} C_VEL
LIN {X 0,Y 361.815,Z 334.42,A -85,B 0,C 180,E1 -12907.212,E2 -12907.212} C_VEL
LIN {X 0,Y 361.854,Z 334.412,A -85,B 0,C 180,E1 -12909.861,E2 -12909.861} C_VEL
LIN {X 0,Y 361.836,Z 334.41,A -85,B 0,C 180,E1 -12912.828,E2 -12912.828} C_VEL
LIN {X 0,Y 361.813,Z 334.415,A -85,B 0,C 180,E1 -12915.947,E2 -12915.947} C_VEL
LIN {X 0,Y 361.808,Z 334.417,A -85,B 0,C 180,E1 -12919.249,E2 -12919.249} C_VEL
LIN {X 0,Y 361.863,Z 334.409,A -85,B 0,C 180,E1 -12922.981,E2 -12922.981} C_VEL
LIN {X 0,Y 361.857,Z 334.408,A -85,B 0,C 180,E1 -12926.63,E2 -12926.63} C_VEL
LIN {X 0,Y 361.854,Z 334.409,A -85,B 0,C 180,E1 -12929.67,E2 -12929.67} C_VEL
LIN {X 0,Y 361.86,Z 334.409,A -85,B 0,C 180,E1 -12933.467,E2 -12933.467} C_VEL
LIN {X 0,Y 361.875,Z 334.409,A -85,B 0,C 180,E1 -12937.144,E2 -12937.144} C_VEL
LIN {X 0,Y 361.904,Z 334.406,A -85,B 0,C 180,E1 -12940.723,E2 -12940.723} C_VEL
LIN {X 0,Y 361.929,Z 334.402,A -85,B 0,C 180,E1 -12943.066,E2 -12943.066} C_VEL
LIN {X 0,Y 361.996,Z 334.394,A -85,B 0,C 180,E1 -12946.528,E2 -12946.528} C_VEL
LIN {X 0,Y 362.028,Z 334.386,A -85,B 0,C 180,E1 -12949.938,E2 -12949.938} C_VEL
LIN {X 0,Y 362.143,Z 334.374,A -85,B 0,C 180,E1 -12952.192,E2 -12952.192} C_VEL
LIN {X 0,Y 362.115,Z 334.381,A -85,B 0,C 180,E1 -12954.431,E2 -12954.431} C_VEL
LIN {X 0,Y 362.276,Z 334.356,A -85,B 0,C 180,E1 -12957.776,E2 -12957.776} C_VEL
LIN {X 0,Y 362.354,Z 334.348,A -85,B 0,C 180,E1 -12960,E2 -12960} C_VEL
LIN {X 0,Y 362.276,Z 334.361,A -85,B 0,C 180,E1 -12962.224,E2 -12962.224} C_VEL
LIN {X 0,Y 362.159,Z 334.371,A -85,B 0,C 180,E1 -12966.686,E2 -12966.686} C_VEL
LIN {X 0,Y 362.028,Z 334.392,A -85,B 0,C 180,E1 -12970.062,E2 -12970.062} C_VEL
LIN {X 0,Y 361.995,Z 334.396,A -85,B 0,C 180,E1 -12973.899,E2 -12973.899} C_VEL
LIN {X 0,Y 361.965,Z 334.399,A -85,B 0,C 180,E1 -12977.939,E2 -12977.939} C_VEL
LIN {X 0,Y 361.878,Z 334.41,A -85,B 0,C 180,E1 -12981.654,E2 -12981.654} C_VEL
LIN {X 0,Y 361.881,Z 334.407,A -85,B 0,C 180,E1 -12985.294,E2 -12985.294} C_VEL
LIN {X 0,Y 361.853,Z 334.409,A -85,B 0,C 180,E1 -12989.074,E2 -12989.074} C_VEL
LIN {X 0,Y 361.846,Z 334.41,A -85,B 0,C 180,E1 -12992.945,E2 -12992.945} C_VEL
LIN {X 0,Y 361.866,Z 334.41,A -85,B 0,C 180,E1 -12995.637,E2 -12995.637} C_VEL
LIN {X 0,Y 361.825,Z 334.415,A -85,B 0,C 180,E1 -12999.018,E2 -12999.018} C_VEL
LIN {X 0,Y 361.827,Z 334.414,A -85,B 0,C 180,E1 -13002.83,E2 -13002.83} C_VEL
LIN {X 0,Y 361.872,Z 334.463,A -85,B 0,C 180,E1 -13006.58,E2 -13006.58} C_VEL
LIN {X 0,Y 362.792,Z 339.693,A -85,B 0,C 180,E1 -13010.263,E2 -13010.263} C_VEL
LIN {X 0,Y 363.33,Z 344.082,A -85,B 0,C 180,E1 -13013.156,E2 -13013.156} C_VEL
LIN {X 0,Y 363.269,Z 348.478,A -85,B 0,C 180,E1 -13015.872,E2 -13015.872} C_VEL
LIN {X 0,Y 362.792,Z 353.981,A -85,B 0,C 180,E1 -13019.112,E2 -13019.112} C_VEL
LIN {X 0,Y 362.087,Z 361.212,A -85,B 0,C 180,E1 -13023.234,E2 -13023.234} C_VEL
LIN {X 0,Y 361.626,Z 367.131,A -85,B 0,C 180,E1 -13026.54,E2 -13026.54} C_VEL
LIN {X 0,Y 361.272,Z 373.349,A -85,B 0,C 180,E1 -13029.93,E2 -13029.93} C_VEL
LIN {X 0,Y 363.952,Z 386.817,A -85,B 0,C 180,E1 -13030.56,E2 -13030.56} C_VEL
LIN {X 0,Y 365.856,Z 399.204,A -85,B 0,C 180,E1 -13031.334,E2 -13031.334} C_VEL
LIN {X 0,Y 366.877,Z 408.674,A -85,B 0,C 180,E1 -13032.056,E2 -13032.056} C_VEL
LIN {X 0,Y 365.777,Z 420.863,A -85,B 0,C 180,E1 -13033.105,E2 -13033.105} C_VEL
LIN {X 0,Y 364.646,Z 432.118,A -85,B 0,C 180,E1 -13034.346,E2 -13034.346} C_VEL
LIN {X 0,Y 363.588,Z 442.088,A -85,B 0,C 180,E1 -13035.732,E2 -13035.732} C_VEL
LIN {X 0,Y 362.565,Z 451.759,A -85,B 0,C 180,E1 -13037.404,E2 -13037.404} C_VEL
LIN {X 0,Y 361.718,Z 459.457,A -85,B 0,C 180,E1 -13039.08,E2 -13039.08} C_VEL
LIN {X 0,Y 361.043,Z 466.559,A -85,B 0,C 180,E1 -13041.041,E2 -13041.041} C_VEL
LIN {X 0,Y 360.683,Z 471.286,A -85,B 0,C 180,E1 -13042.723,E2 -13042.723} C_VEL
LIN {X 0,Y 360.43,Z 474.898,A -85,B 0,C 180,E1 -13044.405,E2 -13044.405} C_VEL
LIN {X 0,Y 360.386,Z 476.763,A -85,B 0,C 180,E1 -13045.526,E2 -13045.526} C_VEL
LIN {X 0,Y 360.303,Z 478.161,A -85,B 0,C 180,E1 -13046.645,E2 -13046.645} C_VEL
LIN {X 0,Y 360.293,Z 479.769,A -85,B 0,C 180,E1 -13048.882,E2 -13048.882} C_VEL
LIN {X 0,Y 360.315,Z 479.986,A -85,B 0,C 180,E1 -13050,E2 -13050} C_VEL
LIN {X 0,Y 360.293,Z 479.768,A -85,B 0,C 180,E1 -13051.117,E2 -13051.117} C_VEL
LIN {X 0,Y 360.302,Z 478.161,A -85,B 0,C 180,E1 -13053.354,E2 -13053.354} C_VEL
LIN {X 0,Y 360.385,Z 476.763,A -85,B 0,C 180,E1 -13054.473,E2 -13054.473} C_VEL
LIN {X 0,Y 360.462,Z 473.95,A -85,B 0,C 180,E1 -13056.087,E2 -13056.087} C_VEL
LIN {X 0,Y 360.734,Z 469.84,A -85,B 0,C 180,E1 -13057.838,E2 -13057.838} C_VEL
LIN {X 0,Y 361.293,Z 463.724,A -85,B 0,C 180,E1 -13059.799,E2 -13059.799} C_VEL
LIN {X 0,Y 361.938,Z 457.041,A -85,B 0,C 180,E1 -13061.48,E2 -13061.48} C_VEL
LIN {X 0,Y 362.906,Z 448.756,A -85,B 0,C 180,E1 -13063.152,E2 -13063.152} C_VEL
LIN {X 0,Y 363.818,Z 440.264,A -85,B 0,C 180,E1 -13064.543,E2 -13064.543} C_VEL
LIN {X 0,Y 364.844,Z 429.769,A -85,B 0,C 180,E1 -13065.931,E2 -13065.931} C_VEL
LIN {X 0,Y 365.877,Z 419.391,A -85,B 0,C 180,E1 -13067.033,E2 -13067.033} C_VEL
LIN {X 0,Y 366.871,Z 408.623,A -85,B 0,C 180,E1 -13067.943,E2 -13067.943} C_VEL
LIN {X 0,Y 365.675,Z 397.794,A -85,B 0,C 180,E1 -13068.759,E2 -13068.759} C_VEL
LIN {X 0,Y 363.661,Z 385.259,A -85,B 0,C 180,E1 -13069.518,E2 -13069.518} C_VEL
LIN {X 0,Y 361.253,Z 373.185,A -85,B 0,C 180,E1 -13070.089,E2 -13070.089} C_VEL
LIN {X 0,Y 361.742,Z 366,A -85,B 0,C 180,E1 -13074.078,E2 -13074.078} C_VEL
LIN {X 0,Y 362.231,Z 359.464,A -85,B 0,C 180,E1 -13077.751,E2 -13077.751} C_VEL
LIN {X 0,Y 362.854,Z 352.83,A -85,B 0,C 180,E1 -13081.546,E2 -13081.546} C_VEL
LIN {X 0,Y 363.348,Z 347.34,A -85,B 0,C 180,E1 -13084.791,E2 -13084.791} C_VEL
LIN {X 0,Y 363.26,Z 342.999,A -85,B 0,C 180,E1 -13087.512,E2 -13087.512} C_VEL
LIN {X 0,Y 362.551,Z 337.985,A -85,B 0,C 180,E1 -13090.886,E2 -13090.886} C_VEL
LIN {X 0,Y 361.921,Z 334.41,A -85,B 0,C 180,E1 -13093.578,E2 -13093.578} C_VEL
LIN {X 0,Y 361.825,Z 334.412,A -85,B 0,C 180,E1 -13097.568,E2 -13097.568} C_VEL
LIN {X 0,Y 361.839,Z 334.41,A -85,B 0,C 180,E1 -13101.571,E2 -13101.571} C_VEL
LIN {X 0,Y 361.868,Z 334.412,A -85,B 0,C 180,E1 -13104.654,E2 -13104.654} C_VEL
LIN {X 0,Y 361.83,Z 334.415,A -85,B 0,C 180,E1 -13108.37,E2 -13108.37} C_VEL
LIN {X 0,Y 361.858,Z 334.409,A -85,B 0,C 180,E1 -13110.951,E2 -13110.951} C_VEL
LIN {X 0,Y 361.875,Z 334.408,A -85,B 0,C 180,E1 -13114.706,E2 -13114.706} C_VEL
LIN {X 0,Y 361.873,Z 334.411,A -85,B 0,C 180,E1 -13118.346,E2 -13118.346} C_VEL
LIN {X 0,Y 361.959,Z 334.4,A -85,B 0,C 180,E1 -13122.061,E2 -13122.061} C_VEL
LIN {X 0,Y 361.989,Z 334.397,A -85,B 0,C 180,E1 -13126.101,E2 -13126.101} C_VEL
LIN {X 0,Y 362.022,Z 334.393,A -85,B 0,C 180,E1 -13129.938,E2 -13129.938} C_VEL
LIN {X 0,Y 362.142,Z 334.375,A -85,B 0,C 180,E1 -13132.192,E2 -13132.192} C_VEL
LIN {X 0,Y 362.115,Z 334.376,A -85,B 0,C 180,E1 -13134.431,E2 -13134.431} C_VEL
LIN {X 0,Y 362.273,Z 334.362,A -85,B 0,C 180,E1 -13137.776,E2 -13137.776} C_VEL
LIN {X 0,Y 362.35,Z 334.349,A -85,B 0,C 180,E1 -13140,E2 -13140} C_VEL
LIN {X 0,Y 362.271,Z 334.357,A -85,B 0,C 180,E1 -13142.224,E2 -13142.224} C_VEL
LIN {X 0,Y 362.164,Z 334.369,A -85,B 0,C 180,E1 -13146.686,E2 -13146.686} C_VEL
LIN {X 0,Y 362.065,Z 334.383,A -85,B 0,C 180,E1 -13148.934,E2 -13148.934} C_VEL
LIN {X 0,Y 361.95,Z 334.395,A -85,B 0,C 180,E1 -13152.333,E2 -13152.333} C_VEL
LIN {X 0,Y 361.952,Z 334.396,A -85,B 0,C 180,E1 -13154.621,E2 -13154.621} C_VEL
LIN {X 0,Y 361.947,Z 334.396,A -85,B 0,C 180,E1 -13158.1,E2 -13158.1} C_VEL
LIN {X 0,Y 361.881,Z 334.405,A -85,B 0,C 180,E1 -13161.654,E2 -13161.654} C_VEL
LIN {X 0,Y 361.875,Z 334.408,A -85,B 0,C 180,E1 -13165.294,E2 -13165.294} C_VEL
LIN {X 0,Y 361.848,Z 334.413,A -85,B 0,C 180,E1 -13169.074,E2 -13169.074} C_VEL
LIN {X 0,Y 361.842,Z 334.414,A -85,B 0,C 180,E1 -13172.946,E2 -13172.946} C_VEL
LIN {X 0,Y 361.861,Z 334.407,A -85,B 0,C 180,E1 -13175.638,E2 -13175.638} C_VEL
LIN {X 0,Y 361.82,Z 334.414,A -85,B 0,C 180,E1 -13179.019,E2 -13179.019} C_VEL
LIN {X 0,Y 361.827,Z 334.414,A -85,B 0,C 180,E1 -13182.83,E2 -13182.83} C_VEL
LIN {X 0,Y 361.821,Z 334.413,A -85,B 0,C 180,E1 -13185.947,E2 -13185.947} C_VEL
LIN {X 0,Y 361.869,Z 334.406,A -85,B 0,C 180,E1 -13189.239,E2 -13189.239} C_VEL
LIN {X 0,Y 361.858,Z 334.408,A -85,B 0,C 180,E1 -13191.575,E2 -13191.575} C_VEL
LIN {X 0,Y 361.812,Z 334.42,A -85,B 0,C 180,E1 -13192.977,E2 -13192.977} C_VEL
LIN {X 0,Y 361.827,Z 335.789,A -85,B 0,C 180,E1 -13194.666,E2 -13194.666} C_VEL
LIN {X 0,Y 361.756,Z 338.399,A -85,B 0,C 180,E1 -13197.047,E2 -13197.047} C_VEL
LIN {X 0,Y 361.591,Z 341.303,A -85,B 0,C 180,E1 -13199.647,E2 -13199.647} C_VEL
LIN {X 0,Y 361.303,Z 345.757,A -85,B 0,C 180,E1 -13203.481,E2 -13203.481} C_VEL
LIN {X 0,Y 361.058,Z 350.132,A -85,B 0,C 180,E1 -13207.09,E2 -13207.09} C_VEL
LIN {X 0,Y 360.973,Z 353.923,A -85,B 0,C 180,E1 -13209.997,E2 -13209.997} C_VEL
LIN {X 0,Y 364.367,Z 367.063,A -85,B 0,C 180,E1 -13210.691,E2 -13210.691} C_VEL
LIN {X 0,Y 367.078,Z 380.22,A -85,B 0,C 180,E1 -13211.588,E2 -13211.588} C_VEL
LIN {X 0,Y 367.557,Z 384.71,A -85,B 0,C 180,E1 -13211.933,E2 -13211.933} C_VEL
LIN {X 0,Y 366.619,Z 396.226,A -85,B 0,C 180,E1 -13212.859,E2 -13212.859} C_VEL
LIN {X 0,Y 365.628,Z 406.925,A -85,B 0,C 180,E1 -13213.964,E2 -13213.964} C_VEL
LIN {X 0,Y 364.726,Z 416.604,A -85,B 0,C 180,E1 -13215.208,E2 -13215.208} C_VEL
LIN {X 0,Y 363.663,Z 425.443,A -85,B 0,C 180,E1 -13216.591,E2 -13216.591} C_VEL
LIN {X 0,Y 362.702,Z 434.06,A -85,B 0,C 180,E1 -13218.262,E2 -13218.262} C_VEL
LIN {X 0,Y 361.909,Z 440.928,A -85,B 0,C 180,E1 -13219.935,E2 -13219.935} C_VEL
LIN {X 0,Y 361.277,Z 446.427,A -85,B 0,C 180,E1 -13221.611,E2 -13221.611} C_VEL
LIN {X 0,Y 360.847,Z 451.647,A -85,B 0,C 180,E1 -13223.703,E2 -13223.703} C_VEL
LIN {X 0,Y 360.562,Z 454.88,A -85,B 0,C 180,E1 -13225.529,E2 -13225.529} C_VEL
LIN {X 0,Y 360.422,Z 456.278,A -85,B 0,C 180,E1 -13226.647,E2 -13226.647} C_VEL
LIN {X 0,Y 360.368,Z 457.882,A -85,B 0,C 180,E1 -13228.883,E2 -13228.883} C_VEL
LIN {X 0,Y 360.362,Z 458.113,A -85,B 0,C 180,E1 -13230,E2 -13230} C_VEL
LIN {X 0,Y 360.368,Z 457.923,A -85,B 0,C 180,E1 -13231.118,E2 -13231.118} C_VEL
LIN {X 0,Y 360.42,Z 456.374,A -85,B 0,C 180,E1 -13233.354,E2 -13233.354} C_VEL
LIN {X 0,Y 360.559,Z 455.017,A -85,B 0,C 180,E1 -13234.472,E2 -13234.472} C_VEL
LIN {X 0,Y 360.847,Z 451.865,A -85,B 0,C 180,E1 -13236.296,E2 -13236.296} C_VEL
LIN {X 0,Y 361.119,Z 448.268,A -85,B 0,C 180,E1 -13237.83,E2 -13237.83} C_VEL
LIN {X 0,Y 361.647,Z 443.255,A -85,B 0,C 180,E1 -13239.508,E2 -13239.508} C_VEL
LIN {X 0,Y 362.357,Z 436.942,A -85,B 0,C 180,E1 -13241.184,E2 -13241.184} C_VEL
LIN {X 0,Y 363.258,Z 429.039,A -85,B 0,C 180,E1 -13242.856,E2 -13242.856} C_VEL
LIN {X 0,Y 364.445,Z 419.204,A -85,B 0,C 180,E1 -13244.519,E2 -13244.519} C_VEL
LIN {X 0,Y 365.388,Z 409.892,A -85,B 0,C 180,E1 -13245.784,E2 -13245.784} C_VEL
LIN {X 0,Y 366.362,Z 398.658,A -85,B 0,C 180,E1 -13247.01,E2 -13247.01} C_VEL
LIN {X 0,Y 367.455,Z 386.913,A -85,B 0,C 180,E1 -13248.008,E2 -13248.008} C_VEL
LIN {X 0,Y 367.55,Z 383.095,A -85,B 0,C 180,E1 -13248.287,E2 -13248.287} C_VEL
LIN {X 0,Y 365.184,Z 370.757,A -85,B 0,C 180,E1 -13249.186,E2 -13249.186} C_VEL
LIN {X 0,Y 362.042,Z 358.142,A -85,B 0,C 180,E1 -13249.909,E2 -13249.909} C_VEL
LIN {X 0,Y 360.949,Z 353.764,A -85,B 0,C 180,E1 -13250.142,E2 -13250.142} C_VEL
LIN {X 0,Y 361.141,Z 348.787,A -85,B 0,C 180,E1 -13254.121,E2 -13254.121} C_VEL
LIN {X 0,Y 361.395,Z 344.359,A -85,B 0,C 180,E1 -13257.822,E2 -13257.822} C_VEL
LIN {X 0,Y 361.676,Z 339.949,A -85,B 0,C 180,E1 -13261.645,E2 -13261.645} C_VEL
LIN {X 0,Y 361.771,Z 338.475,A -85,B 0,C 180,E1 -13262.962,E2 -13262.962} C_VEL
LIN {X 0,Y 361.131,Z 337.569,A -85,B 0,C 180,E1 -13263.881,E2 -13263.881} C_VEL
LIN {X 0,Y 358.284,Z 336.375,A -85,B 0,C 180,E1 -13265.381,E2 -13265.381} C_VEL
LIN {X 0,Y 355.87,Z 335.626,A -85,B 0,C 180,E1 -13266.601,E2 -13266.601} C_VEL
LIN {X 0,Y 354.855,Z 335.319,A -85,B 0,C 180,E1 -13267.547,E2 -13267.547} C_VEL
LIN {X 0,Y 354.785,Z 335.294,A -85,B 0,C 180,E1 -13267.868,E2 -13267.868} C_VEL
LIN {X 0,Y 354.787,Z 335.29,A -85,B 0,C 180,E1 -13271.171,E2 -13271.171} C_VEL
LIN {X 0,Y 354.761,Z 335.292,A -85,B 0,C 180,E1 -13274.506,E2 -13274.506} C_VEL
LIN {X 0,Y 354.78,Z 335.293,A -85,B 0,C 180,E1 -13277.66,E2 -13277.66} C_VEL
LIN {X 0,Y 354.784,Z 335.289,A -85,B 0,C 180,E1 -13280.662,E2 -13280.662} C_VEL
LIN {X 0,Y 354.82,Z 335.284,A -85,B 0,C 180,E1 -13284.3,E2 -13284.3} C_VEL
LIN {X 0,Y 354.785,Z 335.29,A -85,B 0,C 180,E1 -13287.666,E2 -13287.666} C_VEL
LIN {X 0,Y 354.797,Z 335.288,A -85,B 0,C 180,E1 -13291.614,E2 -13291.614} C_VEL
LIN {X 0,Y 354.832,Z 335.283,A -85,B 0,C 180,E1 -13295.657,E2 -13295.657} C_VEL
LIN {X 0,Y 354.824,Z 335.287,A -85,B 0,C 180,E1 -13299.113,E2 -13299.113} C_VEL
LIN {X 0,Y 354.895,Z 335.28,A -85,B 0,C 180,E1 -13302.72,E2 -13302.72} C_VEL
LIN {X 0,Y 354.948,Z 335.27,A -85,B 0,C 180,E1 -13306.255,E2 -13306.255} C_VEL
LIN {X 0,Y 354.975,Z 335.265,A -85,B 0,C 180,E1 -13309.736,E2 -13309.736} C_VEL
LIN {X 0,Y 355.126,Z 335.247,A -85,B 0,C 180,E1 -13312.037,E2 -13312.037} C_VEL
LIN {X 0,Y 355.089,Z 335.254,A -85,B 0,C 180,E1 -13314.321,E2 -13314.321} C_VEL
LIN {X 0,Y 355.24,Z 335.232,A -85,B 0,C 180,E1 -13317.732,E2 -13317.732} C_VEL
LIN {X 0,Y 355.306,Z 335.226,A -85,B 0,C 180,E1 -13320,E2 -13320} C_VEL
LIN {X 0,Y 355.239,Z 335.238,A -85,B 0,C 180,E1 -13322.268,E2 -13322.268} C_VEL
LIN {X 0,Y 355.123,Z 335.247,A -85,B 0,C 180,E1 -13326.819,E2 -13326.819} C_VEL
LIN {X 0,Y 354.974,Z 335.269,A -85,B 0,C 180,E1 -13330.264,E2 -13330.264} C_VEL
LIN {X 0,Y 354.94,Z 335.275,A -85,B 0,C 180,E1 -13334.019,E2 -13334.019} C_VEL
LIN {X 0,Y 354.92,Z 335.275,A -85,B 0,C 180,E1 -13338.108,E2 -13338.108} C_VEL
LIN {X 0,Y 354.824,Z 335.286,A -85,B 0,C 180,E1 -13342.107,E2 -13342.107} C_VEL
LIN {X 0,Y 354.812,Z 335.289,A -85,B 0,C 180,E1 -13345.834,E2 -13345.834} C_VEL
LIN {X 0,Y 354.794,Z 335.292,A -85,B 0,C 180,E1 -13349.684,E2 -13349.684} C_VEL
LIN {X 0,Y 354.785,Z 335.289,A -85,B 0,C 180,E1 -13352.334,E2 -13352.334} C_VEL
